  Call Extruder(8.25300)
  MoveL 4700 to (-39.1, 156.17, 78.65) mm, rotated rx -180 ry 0 rz 180 deg; joints [-141.891, 64.538, -73.427, 141.555, 83.016, 5.514]
  MoveL 4701 to (-39.1, 156.17, 78.65) mm, rotated rx -180 ry 0 rz 180 deg; joints [-141.891, 64.538, -73.427, 141.555, 83.016, 5.514]
  Call Extruder(8.43572)
  MoveL 4702 to (-39.22, 155.87, 78.65) mm, rotated rx -180 ry 0 rz 180 deg; joints [-141.96, 64.533, -73.433, 141.623, 83.001, 5.512]
  MoveL 4703 to (-39.22, 155.87, 78.65) mm, rotated rx -180 ry 0 rz 180 deg; joints [-141.96, 64.533, -73.433, 141.623, 83.001, 5.512]
  Call Extruder(8.61768)
  MoveL 4704 to (-39.35, 155.58, 78.65) mm, rotated rx -180 ry 0 rz 180 deg; joints [-142.029, 64.528, -73.439, 141.691, 82.986, 5.51]
  MoveL 4705 to (-39.35, 155.58, 78.65) mm, rotated rx -180 ry 0 rz 180 deg; joints [-142.029, 64.528, -73.439, 141.691, 82.986, 5.51]
  Call Extruder(8.76501)
  MoveL 4706 to (-39.44, 155.34, 78.65) mm, rotated rx -180 ry 0 rz 180 deg; joints [-142.085, 64.524, -73.444, 141.746, 82.973, 5.509]
  MoveL 4707 to (-39.44, 155.34, 78.65) mm, rotated rx -180 ry 0 rz 180 deg; joints [-142.085, 64.524, -73.444, 141.746, 82.973, 5.509]
  Call Extruder(8.87825)
  MoveL 4708 to (-39.5, 155.15, 78.65) mm, rotated rx -180 ry 0 rz 180 deg; joints [-142.127, 64.52, -73.449, 141.788, 82.963, 5.509]
  MoveL 4709 to (-39.5, 155.15, 78.65) mm, rotated rx -180 ry 0 rz 180 deg; joints [-142.127, 64.52, -73.449, 141.788, 82.963, 5.509]
  Call Extruder(8.99103)
  MoveL 4710 to (-39.56, 154.97, 78.65) mm, rotated rx -180 ry 0 rz 180 deg; joints [-142.169, 64.516, -73.453, 141.83, 82.952, 5.509]
  MoveL 4711 to (-39.56, 154.97, 78.65) mm, rotated rx -180 ry 0 rz 180 deg; joints [-142.169, 64.516, -73.453, 141.83, 82.952, 5.509]
  Call Extruder(9.10338)
  MoveL 4712 to (-39.62, 154.78, 78.65) mm, rotated rx 180 ry 0 rz 180 deg; joints [-142.212, 64.512, -73.458, 141.872, 82.941, 5.509]
  MoveL 4713 to (-39.62, 154.78, 78.65) mm, rotated rx 180 ry 0 rz 180 deg; joints [-142.212, 64.512, -73.458, 141.872, 82.941, 5.509]
  Call Extruder(9.21528)
  MoveL 4714 to (-39.68, 154.59, 78.65) mm, rotated rx 180 ry 0 rz -180 deg; joints [-142.254, 64.508, -73.462, 141.913, 82.931, 5.509]
  MoveL 4715 to (-39.68, 154.59, 78.65) mm, rotated rx 180 ry 0 rz -180 deg; joints [-142.254, 64.508, -73.462, 141.913, 82.931, 5.509]
  Call Extruder(9.33668)
  MoveL 4716 to (-39.75, 154.38, 78.65) mm, rotated rx 180 ry 0 rz 180 deg; joints [-142.3, 64.504, -73.467, 141.959, 82.919, 5.509]
  MoveL 4717 to (-39.75, 154.38, 78.65) mm, rotated rx 180 ry 0 rz 180 deg; joints [-142.3, 64.504, -73.467, 141.959, 82.919, 5.509]
  Call Extruder(9.46748)
  MoveL 4718 to (-39.81, 154.16, 78.65) mm, rotated rx -180 ry 0 rz 180 deg; joints [-142.35, 64.499, -73.473, 142.008, 82.906, 5.51]
  MoveL 4719 to (-39.81, 154.16, 78.65) mm, rotated rx -180 ry 0 rz 180 deg; joints [-142.35, 64.499, -73.473, 142.008, 82.906, 5.51]
  Call Extruder(9.59770)
  MoveL 4720 to (-39.88, 153.94, 78.65) mm, rotated rx 180 ry 0 rz 180 deg; joints [-142.399, 64.494, -73.478, 142.056, 82.893, 5.51]
  MoveL 4721 to (-39.88, 153.94, 78.65) mm, rotated rx 180 ry 0 rz 180 deg; joints [-142.399, 64.494, -73.478, 142.056, 82.893, 5.51]
  Call Extruder(9.72737)
  MoveL 4722 to (-39.95, 153.71, 78.65) mm, rotated rx -180 ry 0 rz 180 deg; joints [-142.449, 64.49, -73.484, 142.106, 82.88, 5.51]
  MoveL 4723 to (-39.95, 153.71, 78.65) mm, rotated rx -180 ry 0 rz 180 deg; joints [-142.449, 64.49, -73.484, 142.106, 82.88, 5.51]
  Call Extruder(9.85647)
  MoveL 4724 to (-40.02, 153.49, 78.65) mm, rotated rx 180 ry 0 rz -180 deg; joints [-142.498, 64.485, -73.49, 142.155, 82.867, 5.511]
  MoveL 4725 to (-40.02, 153.49, 78.65) mm, rotated rx 180 ry 0 rz -180 deg; joints [-142.498, 64.485, -73.49, 142.155, 82.867, 5.511]
  Call Extruder(9.97156)
  MoveL 4726 to (-40.06, 153.28, 78.65) mm, rotated rx 180 ry 0 rz 180 deg; joints [-142.541, 64.48, -73.496, 142.197, 82.854, 5.512]
  MoveL 4727 to (-40.06, 153.28, 78.65) mm, rotated rx 180 ry 0 rz 180 deg; joints [-142.541, 64.48, -73.496, 142.197, 82.854, 5.512]
  Call Extruder(10.08619)
  MoveL 4728 to (-40.11, 153.08, 78.65) mm, rotated rx -180 ry 0 rz 180 deg; joints [-142.584, 64.475, -73.501, 142.239, 82.841, 5.513]
  MoveL 4729 to (-40.11, 153.08, 78.65) mm, rotated rx -180 ry 0 rz 180 deg; joints [-142.584, 64.475, -73.501, 142.239, 82.841, 5.513]
  Call Extruder(10.20037)
  MoveL 4730 to (-40.15, 152.88, 78.65) mm, rotated rx -180 ry 0 rz 180 deg; joints [-142.627, 64.469, -73.507, 142.281, 82.829, 5.515]
  MoveL 4731 to (-40.15, 152.88, 78.65) mm, rotated rx -180 ry 0 rz 180 deg; joints [-142.627, 64.469, -73.507, 142.281, 82.829, 5.515]
  Call Extruder(10.31410)
  MoveL 4732 to (-40.2, 152.67, 78.65) mm, rotated rx -180 ry 0 rz 180 deg; joints [-142.671, 64.464, -73.513, 142.324, 82.816, 5.516]
  MoveL 4733 to (-40.2, 152.67, 78.65) mm, rotated rx -180 ry 0 rz 180 deg; joints [-142.671, 64.464, -73.513, 142.324, 82.816, 5.516]
  Call Extruder(10.43953)
  MoveL 4734 to (-40.24, 152.44, 78.65) mm, rotated rx 180 ry 0 rz 180 deg; joints [-142.718, 64.459, -73.52, 142.371, 82.801, 5.518]
  MoveL 4735 to (-40.24, 152.44, 78.65) mm, rotated rx 180 ry 0 rz 180 deg; joints [-142.718, 64.459, -73.52, 142.371, 82.801, 5.518]
  Call Extruder(10.57650)
  MoveL 4736 to (-40.29, 152.2, 78.65) mm, rotated rx -180 ry 0 rz -180 deg; joints [-142.77, 64.452, -73.527, 142.422, 82.785, 5.52]
  MoveL 4737 to (-40.29, 152.2, 78.65) mm, rotated rx -180 ry 0 rz -180 deg; joints [-142.77, 64.452, -73.527, 142.422, 82.785, 5.52]
  Call Extruder(10.71287)
  MoveL 4738 to (-40.34, 151.95, 78.65) mm, rotated rx 180 ry 0 rz 180 deg; joints [-142.822, 64.446, -73.535, 142.473, 82.769, 5.522]
  MoveL 4739 to (-40.34, 151.95, 78.65) mm, rotated rx 180 ry 0 rz 180 deg; joints [-142.822, 64.446, -73.535, 142.473, 82.769, 5.522]
  Call Extruder(10.84862)
  MoveL 4740 to (-40.39, 151.7, 78.65) mm, rotated rx 180 ry 0 rz 180 deg; joints [-142.874, 64.439, -73.542, 142.524, 82.753, 5.524]
  MoveL 4741 to (-40.39, 151.7, 78.65) mm, rotated rx 180 ry 0 rz 180 deg; joints [-142.874, 64.439, -73.542, 142.524, 82.753, 5.524]
  Call Extruder(10.98377)
  MoveL 4742 to (-40.44, 151.45, 78.65) mm, rotated rx -180 ry 0 rz 180 deg; joints [-142.926, 64.433, -73.55, 142.575, 82.737, 5.526]
  MoveL 4743 to (-40.44, 151.45, 78.65) mm, rotated rx -180 ry 0 rz 180 deg; joints [-142.926, 64.433, -73.55, 142.575, 82.737, 5.526]
  Call Extruder(11.11830)
  MoveL 4744 to (-40.49, 151.2, 78.65) mm, rotated rx -180 ry 0 rz 180 deg; joints [-142.978, 64.426, -73.557, 142.627, 82.721, 5.528]
  MoveL 4745 to (-40.49, 151.2, 78.65) mm, rotated rx -180 ry 0 rz 180 deg; joints [-142.978, 64.426, -73.557, 142.627, 82.721, 5.528]
  Call Extruder(11.25223)
  MoveL 4746 to (-40.54, 150.95, 78.65) mm, rotated rx -180 ry 0 rz 180 deg; joints [-143.031, 64.42, -73.565, 142.678, 82.705, 5.529]
  MoveL 4747 to (-40.54, 150.95, 78.65) mm, rotated rx -180 ry 0 rz 180 deg; joints [-143.031, 64.42, -73.565, 142.678, 82.705, 5.529]
  Call Extruder(11.40008)
  MoveL 4748 to (-40.59, 150.67, 78.65) mm, rotated rx -180 ry 0 rz -180 deg; joints [-143.088, 64.413, -73.573, 142.734, 82.687, 5.532]
  MoveL 4749 to (-40.59, 150.67, 78.65) mm, rotated rx -180 ry 0 rz -180 deg; joints [-143.088, 64.413, -73.573, 142.734, 82.687, 5.532]
  Call Extruder(11.56181)
  MoveL 4750 to (-40.64, 150.37, 78.65) mm, rotated rx 180 ry 0 rz -180 deg; joints [-143.15, 64.404, -73.583, 142.796, 82.667, 5.535]
  MoveL 4751 to (-40.64, 150.37, 78.65) mm, rotated rx 180 ry 0 rz -180 deg; joints [-143.15, 64.404, -73.583, 142.796, 82.667, 5.535]
  Call Extruder(11.72281)
  MoveL 4752 to (-40.69, 150.06, 78.65) mm, rotated rx 180 ry 0 rz -180 deg; joints [-143.213, 64.396, -73.592, 142.857, 82.646, 5.538]
  MoveL 4753 to (-40.69, 150.06, 78.65) mm, rotated rx 180 ry 0 rz -180 deg; joints [-143.213, 64.396, -73.592, 142.857, 82.646, 5.538]
  Call Extruder(11.88308)
  MoveL 4754 to (-40.74, 149.76, 78.65) mm, rotated rx -180 ry 0 rz 180 deg; joints [-143.276, 64.387, -73.602, 142.918, 82.626, 5.541]
  MoveL 4755 to (-40.74, 149.76, 78.65) mm, rotated rx -180 ry 0 rz 180 deg; joints [-143.276, 64.387, -73.602, 142.918, 82.626, 5.541]
  Call Extruder(12.04262)
  MoveL 4756 to (-40.78, 149.45, 78.65) mm, rotated rx -180 ry 0 rz 180 deg; joints [-143.338, 64.379, -73.611, 142.98, 82.605, 5.543]
  MoveL 4757 to (-40.78, 149.45, 78.65) mm, rotated rx -180 ry 0 rz 180 deg; joints [-143.338, 64.379, -73.611, 142.98, 82.605, 5.543]
  Call Extruder(12.20143)
  MoveL 4758 to (-40.83, 149.14, 78.65) mm, rotated rx -180 ry 0 rz 180 deg; joints [-143.401, 64.371, -73.621, 143.042, 82.585, 5.546]
  MoveL 4759 to (-40.83, 149.14, 78.65) mm, rotated rx -180 ry 0 rz 180 deg; joints [-143.401, 64.371, -73.621, 143.042, 82.585, 5.546]
  Call Extruder(12.38010)
  MoveL 4760 to (-40.88, 148.8, 78.65) mm, rotated rx 180 ry 0 rz -180 deg; joints [-143.471, 64.361, -73.632, 143.11, 82.561, 5.55]
  MoveL 4761 to (-40.88, 148.8, 78.65) mm, rotated rx 180 ry 0 rz -180 deg; joints [-143.471, 64.361, -73.632, 143.11, 82.561, 5.55]
  Call Extruder(12.57854)
  MoveL 4762 to (-40.92, 148.41, 78.65) mm, rotated rx -180 ry 0 rz 180 deg; joints [-143.549, 64.349, -73.645, 143.187, 82.535, 5.554]
  MoveL 4763 to (-40.92, 148.41, 78.65) mm, rotated rx -180 ry 0 rz 180 deg; joints [-143.549, 64.349, -73.645, 143.187, 82.535, 5.554]
  Call Extruder(12.77611)
  MoveL 4764 to (-40.97, 148.02, 78.65) mm, rotated rx -180 ry 0 rz -180 deg; joints [-143.627, 64.338, -73.658, 143.263, 82.508, 5.559]
  MoveL 4765 to (-40.97, 148.02, 78.65) mm, rotated rx -180 ry 0 rz -180 deg; joints [-143.627, 64.338, -73.658, 143.263, 82.508, 5.559]
  Call Extruder(12.97282)
  MoveL 4766 to (-41.02, 147.63, 78.65) mm, rotated rx -180 ry 0 rz -180 deg; joints [-143.705, 64.327, -73.671, 143.339, 82.481, 5.563]
  MoveL 4767 to (-41.02, 147.63, 78.65) mm, rotated rx -180 ry 0 rz -180 deg; joints [-143.705, 64.327, -73.671, 143.339, 82.481, 5.563]
  Call Extruder(13.16866)
  MoveL 4768 to (-41.06, 147.25, 78.65) mm, rotated rx -180 ry 0 rz 180 deg; joints [-143.783, 64.316, -73.683, 143.415, 82.454, 5.567]
  MoveL 4769 to (-41.06, 147.25, 78.65) mm, rotated rx -180 ry 0 rz 180 deg; joints [-143.783, 64.316, -73.683, 143.415, 82.454, 5.567]
  Call Extruder(13.46406)
  MoveL 4770 to (-41.11, 146.66, 78.65) mm, rotated rx -180 ry 0 rz -180 deg; joints [-143.899, 64.297, -73.704, 143.529, 82.412, 5.575]
  MoveL 4771 to (-41.11, 146.66, 78.65) mm, rotated rx -180 ry 0 rz -180 deg; joints [-143.899, 64.297, -73.704, 143.529, 82.412, 5.575]
  Call Extruder(13.75812)
  MoveL 4772 to (-41.16, 146.07, 78.65) mm, rotated rx -180 ry 0 rz 180 deg; joints [-144.015, 64.279, -73.724, 143.642, 82.369, 5.583]
  MoveL 4773 to (-41.16, 146.07, 78.65) mm, rotated rx -180 ry 0 rz 180 deg; joints [-144.015, 64.279, -73.724, 143.642, 82.369, 5.583]
  Call Extruder(14.05086)
  MoveL 4774 to (-41.2, 145.48, 78.65) mm, rotated rx -180 ry 0 rz 180 deg; joints [-144.131, 64.261, -73.744, 143.756, 82.327, 5.59]
  MoveL 4775 to (-41.2, 145.48, 78.65) mm, rotated rx -180 ry 0 rz 180 deg; joints [-144.131, 64.261, -73.744, 143.756, 82.327, 5.59]
  Call Extruder(14.62431)
  MoveL 4776 to (-41.25, 144.32, 78.65) mm, rotated rx -180 ry 0 rz -180 deg; joints [-144.355, 64.223, -73.786, 143.975, 82.241, 5.607]
  MoveL 4777 to (-41.25, 144.32, 78.65) mm, rotated rx -180 ry 0 rz -180 deg; joints [-144.355, 64.223, -73.786, 143.975, 82.241, 5.607]
  Call Extruder(15.33827)
  MoveL 4778 to (-41.29, 142.86, 78.65) mm, rotated rx -180 ry 0 rz 180 deg; joints [-144.635, 64.175, -73.839, 144.248, 82.131, 5.629]
  Call Extruder(57.40309)
  MoveL 4779 to (-41.29, 57.14, 78.65) mm, rotated rx -180 ry 0 rz 180 deg; joints [-164.153, 61.724, -76.018, 163.673, 76.26, 3.98]
  Call Extruder(57.83164)
  MoveL 4780 to (-41.27, 56.26, 78.65) mm, rotated rx -180 ry 0 rz 180 deg; joints [-164.382, 61.706, -76.031, 163.906, 76.215, 3.933]
  MoveL 4781 to (-41.27, 56.26, 78.65) mm, rotated rx -180 ry 0 rz 180 deg; joints [-164.382, 61.706, -76.031, 163.906, 76.215, 3.933]
  Call Extruder(58.40509)
  MoveL 4782 to (-41.22, 55.1, 78.65) mm, rotated rx 180 ry 0 rz 180 deg; joints [-164.686, 61.681, -76.049, 164.216, 76.153, 3.87]
  MoveL 4783 to (-41.22, 55.1, 78.65) mm, rotated rx 180 ry 0 rz 180 deg; joints [-164.686, 61.681, -76.049, 164.216, 76.153, 3.87]
  Call Extruder(58.83941)
  MoveL 4784 to (-41.18, 54.23, 78.65) mm, rotated rx 180 ry 0 rz -180 deg; joints [-164.915, 61.662, -76.063, 164.449, 76.105, 3.823]
  MoveL 4785 to (-41.18, 54.23, 78.65) mm, rotated rx 180 ry 0 rz -180 deg; joints [-164.915, 61.662, -76.063, 164.449, 76.105, 3.823]
  Call Extruder(59.13347)
  MoveL 4786 to (-41.13, 53.64, 78.65) mm, rotated rx 180 ry 0 rz 180 deg; joints [-165.068, 61.648, -76.073, 164.605, 76.072, 3.792]
  MoveL 4787 to (-41.13, 53.64, 78.65) mm, rotated rx 180 ry 0 rz 180 deg; joints [-165.068, 61.648, -76.073, 164.605, 76.072, 3.792]
  Call Extruder(59.42887)
  MoveL 4788 to (-41.09, 53.05, 78.65) mm, rotated rx 180 ry 0 rz 180 deg; joints [-165.222, 61.634, -76.083, 164.761, 76.039, 3.76]
  MoveL 4789 to (-41.09, 53.05, 78.65) mm, rotated rx 180 ry 0 rz 180 deg; joints [-165.222, 61.634, -76.083, 164.761, 76.039, 3.76]
  Call Extruder(59.67511)
  MoveL 4790 to (-41.04, 52.56, 78.65) mm, rotated rx 180 ry 0 rz -180 deg; joints [-165.349, 61.622, -76.091, 164.89, 76.011, 3.734]
  MoveL 4791 to (-41.04, 52.56, 78.65) mm, rotated rx 180 ry 0 rz -180 deg; joints [-165.349, 61.622, -76.091, 164.89, 76.011, 3.734]
  Call Extruder(59.87182)
  MoveL 4792 to (-40.99, 52.17, 78.65) mm, rotated rx -180 ry 0 rz 180 deg; joints [-165.449, 61.612, -76.099, 164.993, 75.987, 3.714]
  MoveL 4793 to (-40.99, 52.17, 78.65) mm, rotated rx -180 ry 0 rz 180 deg; joints [-165.449, 61.612, -76.099, 164.993, 75.987, 3.714]
  Call Extruder(60.06939)
  MoveL 4794 to (-40.95, 51.78, 78.65) mm, rotated rx -180 ry 0 rz 180 deg; joints [-165.549, 61.602, -76.106, 165.095, 75.964, 3.694]
  MoveL 4795 to (-40.95, 51.78, 78.65) mm, rotated rx -180 ry 0 rz 180 deg; joints [-165.549, 61.602, -76.106, 165.095, 75.964, 3.694]
  Call Extruder(60.26783)
  MoveL 4796 to (-40.9, 51.4, 78.65) mm, rotated rx 180 ry 0 rz 180 deg; joints [-165.65, 61.592, -76.113, 165.197, 75.941, 3.673]
  MoveL 4797 to (-40.9, 51.4, 78.65) mm, rotated rx 180 ry 0 rz 180 deg; joints [-165.65, 61.592, -76.113, 165.197, 75.941, 3.673]
  Call Extruder(60.46714)
  MoveL 4798 to (-40.86, 51.01, 78.65) mm, rotated rx -180 ry 0 rz -180 deg; joints [-165.751, 61.582, -76.12, 165.299, 75.918, 3.652]
  MoveL 4799 to (-40.86, 51.01, 78.65) mm, rotated rx -180 ry 0 rz -180 deg; joints [-165.751, 61.582, -76.12, 165.299, 75.918, 3.652]
  Call Extruder(60.62596)
  MoveL 4800 to (-40.81, 50.7, 78.65) mm, rotated rx 180 ry 0 rz -180 deg; joints [-165.829, 61.573, -76.126, 165.379, 75.899, 3.637]
  MoveL 4801 to (-40.81, 50.7, 78.65) mm, rotated rx 180 ry 0 rz -180 deg; joints [-165.829, 61.573, -76.126, 165.379, 75.899, 3.637]
  Call Extruder(60.78550)
  MoveL 4802 to (-40.76, 50.4, 78.65) mm, rotated rx 180 ry 0 rz 180 deg; joints [-165.908, 61.564, -76.132, 165.46, 75.88, 3.621]
  MoveL 4803 to (-40.76, 50.4, 78.65) mm, rotated rx 180 ry 0 rz 180 deg; joints [-165.908, 61.564, -76.132, 165.46, 75.88, 3.621]
  Call Extruder(60.94577)
  MoveL 4804 to (-40.71, 50.09, 78.65) mm, rotated rx 180 ry 0 rz 180 deg; joints [-165.987, 61.555, -76.138, 165.54, 75.861, 3.605]
  MoveL 4805 to (-40.71, 50.09, 78.65) mm, rotated rx 180 ry 0 rz 180 deg; joints [-165.987, 61.555, -76.138, 165.54, 75.861, 3.605]
  Call Extruder(61.10677)
  MoveL 4806 to (-40.66, 49.79, 78.65) mm, rotated rx -180 ry 0 rz -180 deg; joints [-166.066, 61.547, -76.144, 165.62, 75.841, 3.589]
  MoveL 4807 to (-40.66, 49.79, 78.65) mm, rotated rx -180 ry 0 rz -180 deg; joints [-166.066, 61.547, -76.144, 165.62, 75.841, 3.589]
  Call Extruder(61.26850)
  MoveL 4808 to (-40.61, 49.48, 78.65) mm, rotated rx 180 ry 0 rz 180 deg; joints [-166.145, 61.538, -76.15, 165.701, 75.822, 3.572]
  MoveL 4809 to (-40.61, 49.48, 78.65) mm, rotated rx 180 ry 0 rz 180 deg; joints [-166.145, 61.538, -76.15, 165.701, 75.822, 3.572]
  Call Extruder(61.43095)
  MoveL 4810 to (-40.57, 49.17, 78.65) mm, rotated rx 180 ry 0 rz -180 deg; joints [-166.224, 61.53, -76.156, 165.781, 75.803, 3.556]
  MoveL 4811 to (-40.57, 49.17, 78.65) mm, rotated rx 180 ry 0 rz -180 deg; joints [-166.224, 61.53, -76.156, 165.781, 75.803, 3.556]
  Call Extruder(61.56487)
  MoveL 4812 to (-40.52, 48.92, 78.65) mm, rotated rx 180 ry 0 rz 180 deg; joints [-166.288, 61.522, -76.161, 165.846, 75.787, 3.543]
  MoveL 4813 to (-40.52, 48.92, 78.65) mm, rotated rx 180 ry 0 rz 180 deg; joints [-166.288, 61.522, -76.161, 165.846, 75.787, 3.543]
  Call Extruder(61.69941)
  MoveL 4814 to (-40.47, 48.68, 78.65) mm, rotated rx -180 ry 0 rz -180 deg; joints [-166.352, 61.514, -76.167, 165.911, 75.77, 3.53]
  MoveL 4815 to (-40.47, 48.68, 78.65) mm, rotated rx -180 ry 0 rz -180 deg; joints [-166.352, 61.514, -76.167, 165.911, 75.77, 3.53]
  Call Extruder(61.83455)
  MoveL 4816 to (-40.42, 48.43, 78.65) mm, rotated rx 180 ry 0 rz -180 deg; joints [-166.416, 61.506, -76.172, 165.976, 75.754, 3.517]
  MoveL 4817 to (-40.42, 48.43, 78.65) mm, rotated rx 180 ry 0 rz -180 deg; joints [-166.416, 61.506, -76.172, 165.976, 75.754, 3.517]
  Call Extruder(61.97031)
  MoveL 4818 to (-40.37, 48.18, 78.65) mm, rotated rx -180 ry 0 rz 180 deg; joints [-166.48, 61.499, -76.177, 166.041, 75.737, 3.504]
  MoveL 4819 to (-40.37, 48.18, 78.65) mm, rotated rx -180 ry 0 rz 180 deg; joints [-166.48, 61.499, -76.177, 166.041, 75.737, 3.504]
  Call Extruder(62.10667)
  MoveL 4820 to (-40.32, 47.93, 78.65) mm, rotated rx -180 ry 0 rz 180 deg; joints [-166.544, 61.491, -76.183, 166.107, 75.721, 3.491]
  MoveL 4821 to (-40.32, 47.93, 78.65) mm, rotated rx -180 ry 0 rz 180 deg; joints [-166.544, 61.491, -76.183, 166.107, 75.721, 3.491]
  Call Extruder(62.24365)
  MoveL 4822 to (-40.27, 47.68, 78.65) mm, rotated rx -180 ry 0 rz 180 deg; joints [-166.608, 61.484, -76.188, 166.172, 75.704, 3.478]
  MoveL 4823 to (-40.27, 47.68, 78.65) mm, rotated rx -180 ry 0 rz 180 deg; joints [-166.608, 61.484, -76.188, 166.172, 75.704, 3.478]
  Call Extruder(62.38124)
  MoveL 4824 to (-40.22, 47.43, 78.65) mm, rotated rx -180 ry 0 rz 180 deg; joints [-166.673, 61.476, -76.193, 166.237, 75.688, 3.465]
  MoveL 4825 to (-40.22, 47.43, 78.65) mm, rotated rx -180 ry 0 rz 180 deg; joints [-166.673, 61.476, -76.193, 166.237, 75.688, 3.465]
  Call Extruder(62.49496)
  MoveL 4826 to (-40.17, 47.23, 78.65) mm, rotated rx -180 ry 0 rz 180 deg; joints [-166.725, 61.47, -76.197, 166.291, 75.674, 3.454]
  MoveL 4827 to (-40.17, 47.23, 78.65) mm, rotated rx -180 ry 0 rz 180 deg; joints [-166.725, 61.47, -76.197, 166.291, 75.674, 3.454]
  Call Extruder(62.60914)
  MoveL 4828 to (-40.13, 47.02, 78.65) mm, rotated rx 180 ry 0 rz 180 deg; joints [-166.778, 61.463, -76.202, 166.344, 75.66, 3.443]
  MoveL 4829 to (-40.13, 47.02, 78.65) mm, rotated rx 180 ry 0 rz 180 deg; joints [-166.778, 61.463, -76.202, 166.344, 75.66, 3.443]
  Call Extruder(62.72378)
  MoveL 4830 to (-40.08, 46.82, 78.65) mm, rotated rx 180 ry 0 rz -180 deg; joints [-166.83, 61.457, -76.206, 166.398, 75.646, 3.433]
  MoveL 4831 to (-40.08, 46.82, 78.65) mm, rotated rx 180 ry 0 rz -180 deg; joints [-166.83, 61.457, -76.206, 166.398, 75.646, 3.433]
  Call Extruder(62.83886)
  MoveL 4832 to (-40.04, 46.61, 78.65) mm, rotated rx -180 ry 0 rz 180 deg; joints [-166.883, 61.45, -76.211, 166.451, 75.633, 3.422]
  MoveL 4833 to (-40.04, 46.61, 78.65) mm, rotated rx -180 ry 0 rz 180 deg; joints [-166.883, 61.45, -76.211, 166.451, 75.633, 3.422]
  Call Extruder(62.96110)
  MoveL 4834 to (-39.98, 46.4, 78.65) mm, rotated rx -180 ry 0 rz -180 deg; joints [-166.937, 61.443, -76.216, 166.507, 75.617, 3.411]
  MoveL 4835 to (-39.98, 46.4, 78.65) mm, rotated rx -180 ry 0 rz -180 deg; joints [-166.937, 61.443, -76.216, 166.507, 75.617, 3.411]
  Call Extruder(63.09076)
  MoveL 4836 to (-39.92, 46.18, 78.65) mm, rotated rx -180 ry 0 rz 180 deg; joints [-166.994, 61.434, -76.222, 166.564, 75.6, 3.4]
  MoveL 4837 to (-39.92, 46.18, 78.65) mm, rotated rx -180 ry 0 rz 180 deg; joints [-166.994, 61.434, -76.222, 166.564, 75.6, 3.4]
  Call Extruder(63.22099)
  MoveL 4838 to (-39.85, 45.95, 78.65) mm, rotated rx -180 ry 0 rz 180 deg; joints [-167.051, 61.426, -76.227, 166.622, 75.583, 3.389]
  MoveL 4839 to (-39.85, 45.95, 78.65) mm, rotated rx -180 ry 0 rz 180 deg; joints [-167.051, 61.426, -76.227, 166.622, 75.583, 3.389]
  Call Extruder(63.35179)
  MoveL 4840 to (-39.78, 45.73, 78.65) mm, rotated rx 180 ry 0 rz -180 deg; joints [-167.107, 61.418, -76.233, 166.68, 75.566, 3.378]
  MoveL 4841 to (-39.78, 45.73, 78.65) mm, rotated rx 180 ry 0 rz -180 deg; joints [-167.107, 61.418, -76.233, 166.68, 75.566, 3.378]
  Call Extruder(63.48315)
  MoveL 4842 to (-39.71, 45.5, 78.65) mm, rotated rx 180 ry 0 rz 180 deg; joints [-167.164, 61.409, -76.239, 166.737, 75.549, 3.366]
  MoveL 4843 to (-39.71, 45.5, 78.65) mm, rotated rx 180 ry 0 rz 180 deg; joints [-167.164, 61.409, -76.239, 166.737, 75.549, 3.366]
  Call Extruder(63.59505)
  MoveL 4844 to (-39.65, 45.32, 78.65) mm, rotated rx -180 ry 0 rz -180 deg; joints [-167.212, 61.402, -76.244, 166.786, 75.534, 3.357]
  MoveL 4845 to (-39.65, 45.32, 78.65) mm, rotated rx -180 ry 0 rz -180 deg; joints [-167.212, 61.402, -76.244, 166.786, 75.534, 3.357]
  Call Extruder(63.70739)
  MoveL 4846 to (-39.59, 45.13, 78.65) mm, rotated rx -180 ry 0 rz -180 deg; joints [-167.26, 61.395, -76.249, 166.834, 75.52, 3.347]
  MoveL 4847 to (-39.59, 45.13, 78.65) mm, rotated rx -180 ry 0 rz -180 deg; joints [-167.26, 61.395, -76.249, 166.834, 75.52, 3.347]
  Call Extruder(63.82018)
  MoveL 4848 to (-39.53, 44.94, 78.65) mm, rotated rx -180 ry 0 rz -180 deg; joints [-167.307, 61.387, -76.254, 166.882, 75.505, 3.338]
  MoveL 4849 to (-39.53, 44.94, 78.65) mm, rotated rx -180 ry 0 rz -180 deg; joints [-167.307, 61.387, -76.254, 166.882, 75.505, 3.338]
  Call Extruder(63.93342)
  MoveL 4850 to (-39.47, 44.75, 78.65) mm, rotated rx 180 ry 0 rz 180 deg; joints [-167.355, 61.38, -76.259, 166.931, 75.49, 3.329]
  MoveL 4851 to (-39.47, 44.75, 78.65) mm, rotated rx 180 ry 0 rz 180 deg; joints [-167.355, 61.38, -76.259, 166.931, 75.49, 3.329]
  Call Extruder(64.04710)
  MoveL 4852 to (-39.41, 44.56, 78.65) mm, rotated rx -180 ry 0 rz 180 deg; joints [-167.403, 61.373, -76.264, 166.98, 75.475, 3.319]
  MoveL 4853 to (-39.41, 44.56, 78.65) mm, rotated rx -180 ry 0 rz 180 deg; joints [-167.403, 61.373, -76.264, 166.98, 75.475, 3.319]
  Call Extruder(64.22906)
  MoveL 4854 to (-39.29, 44.27, 78.65) mm, rotated rx -180 ry 0 rz -180 deg; joints [-167.475, 61.36, -76.272, 167.053, 75.45, 3.305]
  MoveL 4855 to (-39.29, 44.27, 78.65) mm, rotated rx -180 ry 0 rz -180 deg; joints [-167.475, 61.36, -76.272, 167.053, 75.45, 3.305]
  Call Extruder(64.41178)
  MoveL 4856 to (-39.17, 43.98, 78.65) mm, rotated rx -180 ry 0 rz 180 deg; joints [-167.548, 61.346, -76.281, 167.127, 75.424, 3.292]
  MoveL 4857 to (-39.17, 43.98, 78.65) mm, rotated rx -180 ry 0 rz 180 deg; joints [-167.548, 61.346, -76.281, 167.127, 75.424, 3.292]
  Call Extruder(64.58219)
  MoveL 4858 to (-39.05, 43.71, 78.65) mm, rotated rx -180 ry 0 rz -180 deg; joints [-167.615, 61.334, -76.29, 167.195, 75.4, 3.279]
  MoveL 4859 to (-39.05, 43.71, 78.65) mm, rotated rx -180 ry 0 rz -180 deg; joints [-167.615, 61.334, -76.29, 167.195, 75.4, 3.279]
  Call Extruder(64.74017)
  MoveL 4860 to (-38.94, 43.46, 78.65) mm, rotated rx -180 ry 0 rz -180 deg; joints [-167.677, 61.323, -76.297, 167.258, 75.378, 3.267]
  MoveL 4861 to (-38.94, 43.46, 78.65) mm, rotated rx -180 ry 0 rz -180 deg; joints [-167.677, 61.323, -76.297, 167.258, 75.378, 3.267]
  Call Extruder(64.89876)
  MoveL 4862 to (-38.84, 43.21, 78.65) mm, rotated rx 180 ry 0 rz 180 deg; joints [-167.739, 61.311, -76.305, 167.321, 75.356, 3.255]
  MoveL 4863 to (-38.84, 43.21, 78.65) mm, rotated rx 180 ry 0 rz 180 deg; joints [-167.739, 61.311, -76.305, 167.321, 75.356, 3.255]
  Call Extruder(65.10492)
  MoveL 4864 to (-38.66, 42.91, 78.65) mm, rotated rx -180 ry 0 rz -180 deg; joints [-167.813, 61.294, -76.316, 167.395, 75.324, 3.243]
  MoveL 4865 to (-38.66, 42.91, 78.65) mm, rotated rx -180 ry 0 rz -180 deg; joints [-167.813, 61.294, -76.316, 167.395, 75.324, 3.243]
  Call Extruder(65.31187)
  MoveL 4866 to (-38.49, 42.6, 78.65) mm, rotated rx 180 ry 0 rz 180 deg; joints [-167.886, 61.277, -76.328, 167.469, 75.292, 3.23]
  MoveL 4867 to (-38.49, 42.6, 78.65) mm, rotated rx 180 ry 0 rz 180 deg; joints [-167.886, 61.277, -76.328, 167.469, 75.292, 3.23]
  Call Extruder(65.51959)
  MoveL 4868 to (-38.31, 42.3, 78.65) mm, rotated rx 180 ry 0 rz 180 deg; joints [-167.96, 61.26, -76.339, 167.544, 75.26, 3.217]
  MoveL 4869 to (-38.31, 42.3, 78.65) mm, rotated rx 180 ry 0 rz 180 deg; joints [-167.96, 61.26, -76.339, 167.544, 75.26, 3.217]
  Call Extruder(65.72809)
  MoveL 4870 to (-38.14, 41.99, 78.65) mm, rotated rx -180 ry 0 rz -180 deg; joints [-168.033, 61.243, -76.351, 167.618, 75.228, 3.204]
  MoveL 4871 to (-38.14, 41.99, 78.65) mm, rotated rx -180 ry 0 rz -180 deg; joints [-168.033, 61.243, -76.351, 167.618, 75.228, 3.204]
  Call Extruder(65.90765)
  MoveL 4872 to (-37.96, 41.75, 78.65) mm, rotated rx -180 ry 0 rz -180 deg; joints [-168.091, 61.227, -76.361, 167.676, 75.199, 3.195]
  MoveL 4873 to (-37.96, 41.75, 78.65) mm, rotated rx -180 ry 0 rz -180 deg; joints [-168.091, 61.227, -76.361, 167.676, 75.199, 3.195]
  Call Extruder(66.24108)
  MoveL 4874 to (-37.63, 41.3, 78.65) mm, rotated rx -180 ry 0 rz 180 deg; joints [-168.197, 61.196, -76.381, 167.783, 75.144, 3.178]
  MoveL 4875 to (-37.63, 41.3, 78.65) mm, rotated rx -180 ry 0 rz 180 deg; joints [-168.197, 61.196, -76.381, 167.783, 75.144, 3.178]
  Call Extruder(66.57570)
  MoveL 4876 to (-37.3, 40.85, 78.65) mm, rotated rx 180 ry 0 rz -180 deg; joints [-168.304, 61.166, -76.401, 167.89, 75.089, 3.16]
  Call Extruder(67.40363)
  MoveL 4877 to (-36.39, 39.81, 78.65) mm, rotated rx -180 ry 0 rz 180 deg; joints [-168.541, 61.085, -76.454, 168.128, 74.946, 3.125]
  Call Extruder(68.23154)
  MoveL 4878 to (-35.35, 38.9, 78.65) mm, rotated rx -180 ry 0 rz -180 deg; joints [-168.739, 60.997, -76.51, 168.325, 74.793, 3.102]
  Call Extruder(68.39885)
  MoveL 4879 to (-35.13, 38.73, 78.65) mm, rotated rx 180 ry 0 rz 180 deg; joints [-168.773, 60.979, -76.522, 168.358, 74.761, 3.1]
  MoveL 4880 to (-35.13, 38.73, 78.65) mm, rotated rx 180 ry 0 rz 180 deg; joints [-168.773, 60.979, -76.522, 168.358, 74.761, 3.1]
  Call Extruder(68.73227)
  MoveL 4881 to (-34.68, 38.4, 78.65) mm, rotated rx 180 ry 0 rz 180 deg; joints [-168.84, 60.941, -76.546, 168.424, 74.698, 3.094]
  MoveL 4882 to (-34.68, 38.4, 78.65) mm, rotated rx 180 ry 0 rz 180 deg; joints [-168.84, 60.941, -76.546, 168.424, 74.698, 3.094]
  Call Extruder(69.06451)
  MoveL 4883 to (-34.23, 38.08, 78.65) mm, rotated rx -180 ry 0 rz -180 deg; joints [-168.908, 60.904, -76.569, 168.492, 74.634, 3.088]
  MoveL 4884 to (-34.23, 38.08, 78.65) mm, rotated rx -180 ry 0 rz -180 deg; joints [-168.908, 60.904, -76.569, 168.492, 74.634, 3.088]
  Call Extruder(69.18222)
  MoveL 4885 to (-34.05, 37.98, 78.65) mm, rotated rx -180 ry 0 rz -180 deg; joints [-168.927, 60.89, -76.578, 168.51, 74.611, 3.088]
  MoveL 4886 to (-34.05, 37.98, 78.65) mm, rotated rx -180 ry 0 rz -180 deg; joints [-168.927, 60.89, -76.578, 168.51, 74.611, 3.088]
  Call Extruder(69.38994)
  MoveL 4887 to (-33.75, 37.8, 78.65) mm, rotated rx 180 ry 0 rz 180 deg; joints [-168.96, 60.865, -76.593, 168.542, 74.57, 3.087]
  MoveL 4888 to (-33.75, 37.8, 78.65) mm, rotated rx 180 ry 0 rz 180 deg; joints [-168.96, 60.865, -76.593, 168.542, 74.57, 3.087]
  Call Extruder(69.59688)
  MoveL 4889 to (-33.45, 37.63, 78.65) mm, rotated rx -180 ry 0 rz 180 deg; joints [-168.993, 60.84, -76.609, 168.574, 74.529, 3.086]
  MoveL 4890 to (-33.45, 37.63, 78.65) mm, rotated rx -180 ry 0 rz 180 deg; joints [-168.993, 60.84, -76.609, 168.574, 74.529, 3.086]
  Call Extruder(69.80304)
  MoveL 4891 to (-33.14, 37.45, 78.65) mm, rotated rx -180 ry 0 rz -180 deg; joints [-169.026, 60.816, -76.624, 168.606, 74.488, 3.085]
  MoveL 4892 to (-33.14, 37.45, 78.65) mm, rotated rx -180 ry 0 rz -180 deg; joints [-169.026, 60.816, -76.624, 168.606, 74.488, 3.085]
  Call Extruder(69.98473)
  MoveL 4893 to (-32.87, 37.31, 78.65) mm, rotated rx 180 ry 0 rz 180 deg; joints [-169.052, 60.793, -76.638, 168.63, 74.451, 3.085]
  MoveL 4894 to (-32.87, 37.31, 78.65) mm, rotated rx 180 ry 0 rz 180 deg; joints [-169.052, 60.793, -76.638, 168.63, 74.451, 3.085]
  Call Extruder(70.14273)
  MoveL 4895 to (-32.62, 37.2, 78.65) mm, rotated rx 180 ry 0 rz 180 deg; joints [-169.068, 60.774, -76.65, 168.646, 74.419, 3.087]
  MoveL 4896 to (-32.62, 37.2, 78.65) mm, rotated rx 180 ry 0 rz 180 deg; joints [-169.068, 60.774, -76.65, 168.646, 74.419, 3.087]
  Call Extruder(70.30013)
  MoveL 4897 to (-32.37, 37.09, 78.65) mm, rotated rx -180 ry 0 rz 180 deg; joints [-169.085, 60.754, -76.662, 168.662, 74.387, 3.089]
  MoveL 4898 to (-32.37, 37.09, 78.65) mm, rotated rx -180 ry 0 rz 180 deg; joints [-169.085, 60.754, -76.662, 168.662, 74.387, 3.089]
  Call Extruder(70.48284)
  MoveL 4899 to (-32.07, 36.97, 78.65) mm, rotated rx -180 ry 0 rz 180 deg; joints [-169.104, 60.731, -76.676, 168.679, 74.349, 3.092]
  MoveL 4900 to (-32.07, 36.97, 78.65) mm, rotated rx -180 ry 0 rz 180 deg; joints [-169.104, 60.731, -76.676, 168.679, 74.349, 3.092]
  Call Extruder(70.66479)
  MoveL 4901 to (-31.78, 36.85, 78.65) mm, rotated rx -180 ry 0 rz -180 deg; joints [-169.122, 60.708, -76.69, 168.696, 74.312, 3.094]
  MoveL 4902 to (-31.78, 36.85, 78.65) mm, rotated rx -180 ry 0 rz -180 deg; joints [-169.122, 60.708, -76.69, 168.696, 74.312, 3.094]
  Call Extruder(70.81212)
  MoveL 4903 to (-31.54, 36.76, 78.65) mm, rotated rx -180 ry 0 rz -180 deg; joints [-169.135, 60.689, -76.702, 168.708, 74.281, 3.096]
  MoveL 4904 to (-31.54, 36.76, 78.65) mm, rotated rx -180 ry 0 rz -180 deg; joints [-169.135, 60.689, -76.702, 168.708, 74.281, 3.096]
  Call Extruder(70.92535)
  MoveL 4905 to (-31.35, 36.7, 78.65) mm, rotated rx -180 ry 0 rz 180 deg; joints [-169.143, 60.674, -76.711, 168.714, 74.258, 3.099]
  MoveL 4906 to (-31.35, 36.7, 78.65) mm, rotated rx -180 ry 0 rz 180 deg; joints [-169.143, 60.674, -76.711, 168.714, 74.258, 3.099]
  Call Extruder(71.03815)
  MoveL 4907 to (-31.17, 36.64, 78.65) mm, rotated rx -180 ry 0 rz 180 deg; joints [-169.15, 60.659, -76.72, 168.72, 74.234, 3.102]
  MoveL 4908 to (-31.17, 36.64, 78.65) mm, rotated rx -180 ry 0 rz 180 deg; joints [-169.15, 60.659, -76.72, 168.72, 74.234, 3.102]
  Call Extruder(71.15049)
  MoveL 4909 to (-30.98, 36.58, 78.65) mm, rotated rx -180 ry 0 rz 180 deg; joints [-169.157, 60.644, -76.729, 168.726, 74.21, 3.105]
  MoveL 4910 to (-30.98, 36.58, 78.65) mm, rotated rx -180 ry 0 rz 180 deg; joints [-169.157, 60.644, -76.729, 168.726, 74.21, 3.105]
  Call Extruder(71.26240)
  MoveL 4911 to (-30.79, 36.52, 78.65) mm, rotated rx -180 ry 0 rz 180 deg; joints [-169.164, 60.629, -76.737, 168.733, 74.187, 3.107]
  MoveL 4912 to (-30.79, 36.52, 78.65) mm, rotated rx -180 ry 0 rz 180 deg; joints [-169.164, 60.629, -76.737, 168.733, 74.187, 3.107]
  Call Extruder(71.38380)
  MoveL 4913 to (-30.58, 36.45, 78.65) mm, rotated rx 180 ry 0 rz 180 deg; joints [-169.172, 60.613, -76.747, 168.739, 74.161, 3.111]
  MoveL 4914 to (-30.58, 36.45, 78.65) mm, rotated rx 180 ry 0 rz 180 deg; joints [-169.172, 60.613, -76.747, 168.739, 74.161, 3.111]
  Call Extruder(71.51459)
  MoveL 4915 to (-30.36, 36.38, 78.65) mm, rotated rx -180 ry 0 rz -180 deg; joints [-169.179, 60.596, -76.758, 168.745, 74.133, 3.114]
  MoveL 4916 to (-30.36, 36.38, 78.65) mm, rotated rx -180 ry 0 rz -180 deg; joints [-169.179, 60.596, -76.758, 168.745, 74.133, 3.114]
  Call Extruder(71.64481)
  MoveL 4917 to (-30.14, 36.32, 78.65) mm, rotated rx -180 ry 0 rz -180 deg; joints [-169.186, 60.578, -76.768, 168.751, 74.106, 3.118]
  MoveL 4918 to (-30.14, 36.32, 78.65) mm, rotated rx -180 ry 0 rz -180 deg; joints [-169.186, 60.578, -76.768, 168.751, 74.106, 3.118]
  Call Extruder(71.77447)
  MoveL 4919 to (-29.91, 36.25, 78.65) mm, rotated rx -180 ry 0 rz -180 deg; joints [-169.193, 60.561, -76.778, 168.757, 74.078, 3.121]
  MoveL 4920 to (-29.91, 36.25, 78.65) mm, rotated rx -180 ry 0 rz -180 deg; joints [-169.193, 60.561, -76.778, 168.757, 74.078, 3.121]
  Call Extruder(71.90357)
  MoveL 4921 to (-29.69, 36.18, 78.65) mm, rotated rx -180 ry 0 rz -180 deg; joints [-169.201, 60.543, -76.789, 168.763, 74.05, 3.125]
  MoveL 4922 to (-29.69, 36.18, 78.65) mm, rotated rx -180 ry 0 rz -180 deg; joints [-169.201, 60.543, -76.789, 168.763, 74.05, 3.125]
  Call Extruder(72.01864)
  MoveL 4923 to (-29.48, 36.14, 78.65) mm, rotated rx -180 ry 0 rz 180 deg; joints [-169.202, 60.527, -76.798, 168.763, 74.025, 3.13]
  MoveL 4924 to (-29.48, 36.14, 78.65) mm, rotated rx -180 ry 0 rz 180 deg; joints [-169.202, 60.527, -76.798, 168.763, 74.025, 3.13]
  Call Extruder(72.13326)
  MoveL 4925 to (-29.28, 36.09, 78.65) mm, rotated rx -180 ry 0 rz 180 deg; joints [-169.204, 60.512, -76.807, 168.764, 74, 3.134]
  MoveL 4926 to (-29.28, 36.09, 78.65) mm, rotated rx -180 ry 0 rz 180 deg; joints [-169.204, 60.512, -76.807, 168.764, 74, 3.134]
  Call Extruder(72.24743)
  MoveL 4927 to (-29.08, 36.05, 78.65) mm, rotated rx -180 ry 0 rz 180 deg; joints [-169.206, 60.496, -76.817, 168.764, 73.976, 3.139]
  MoveL 4928 to (-29.08, 36.05, 78.65) mm, rotated rx -180 ry 0 rz 180 deg; joints [-169.206, 60.496, -76.817, 168.764, 73.976, 3.139]
  Call Extruder(72.36115)
  MoveL 4929 to (-28.87, 36, 78.65) mm, rotated rx 180 ry 0 rz 180 deg; joints [-169.207, 60.48, -76.826, 168.764, 73.951, 3.144]
  MoveL 4930 to (-28.87, 36, 78.65) mm, rotated rx 180 ry 0 rz 180 deg; joints [-169.207, 60.48, -76.826, 168.764, 73.951, 3.144]
  Call Extruder(72.48657)
  MoveL 4931 to (-28.65, 35.96, 78.65) mm, rotated rx -180 ry 0 rz 180 deg; joints [-169.208, 60.462, -76.836, 168.764, 73.924, 3.149]
  MoveL 4932 to (-28.65, 35.96, 78.65) mm, rotated rx -180 ry 0 rz 180 deg; joints [-169.208, 60.462, -76.836, 168.764, 73.924, 3.149]
  Call Extruder(72.62355)
  MoveL 4933 to (-28.4, 35.91, 78.65) mm, rotated rx -180 ry 0 rz 180 deg; joints [-169.209, 60.443, -76.847, 168.763, 73.894, 3.155]
  MoveL 4934 to (-28.4, 35.91, 78.65) mm, rotated rx -180 ry 0 rz 180 deg; joints [-169.209, 60.443, -76.847, 168.763, 73.894, 3.155]
  Call Extruder(72.75991)
  MoveL 4935 to (-28.15, 35.86, 78.65) mm, rotated rx 180 ry 0 rz 180 deg; joints [-169.21, 60.424, -76.859, 168.762, 73.864, 3.161]
  MoveL 4936 to (-28.15, 35.86, 78.65) mm, rotated rx 180 ry 0 rz 180 deg; joints [-169.21, 60.424, -76.859, 168.762, 73.864, 3.161]
  Call Extruder(72.89567)
  MoveL 4937 to (-27.9, 35.81, 78.65) mm, rotated rx -180 ry 0 rz -180 deg; joints [-169.21, 60.404, -76.87, 168.76, 73.834, 3.167]
  MoveL 4938 to (-27.9, 35.81, 78.65) mm, rotated rx -180 ry 0 rz -180 deg; joints [-169.21, 60.404, -76.87, 168.76, 73.834, 3.167]
  Call Extruder(73.03082)
  MoveL 4939 to (-27.65, 35.76, 78.65) mm, rotated rx -180 ry 0 rz 180 deg; joints [-169.211, 60.385, -76.881, 168.759, 73.804, 3.173]
  MoveL 4940 to (-27.65, 35.76, 78.65) mm, rotated rx -180 ry 0 rz 180 deg; joints [-169.211, 60.385, -76.881, 168.759, 73.804, 3.173]
  Call Extruder(73.16535)
  MoveL 4941 to (-27.4, 35.71, 78.65) mm, rotated rx -180 ry 0 rz -180 deg; joints [-169.212, 60.366, -76.892, 168.758, 73.774, 3.179]
  MoveL 4942 to (-27.4, 35.71, 78.65) mm, rotated rx -180 ry 0 rz -180 deg; joints [-169.212, 60.366, -76.892, 168.758, 73.774, 3.179]
  Call Extruder(73.29928)
  MoveL 4943 to (-27.15, 35.66, 78.65) mm, rotated rx 180 ry 0 rz -180 deg; joints [-169.212, 60.346, -76.903, 168.757, 73.744, 3.185]
  MoveL 4944 to (-27.15, 35.66, 78.65) mm, rotated rx 180 ry 0 rz -180 deg; joints [-169.212, 60.346, -76.903, 168.757, 73.744, 3.185]
  Call Extruder(73.44714)
  MoveL 4945 to (-26.87, 35.61, 78.65) mm, rotated rx -180 ry 0 rz 180 deg; joints [-169.211, 60.325, -76.916, 168.754, 73.711, 3.192]
  MoveL 4946 to (-26.87, 35.61, 78.65) mm, rotated rx -180 ry 0 rz 180 deg; joints [-169.211, 60.325, -76.916, 168.754, 73.711, 3.192]
  Call Extruder(73.60887)
  MoveL 4947 to (-26.57, 35.56, 78.65) mm, rotated rx -180 ry 0 rz 180 deg; joints [-169.208, 60.301, -76.929, 168.749, 73.675, 3.201]
  MoveL 4948 to (-26.57, 35.56, 78.65) mm, rotated rx -180 ry 0 rz 180 deg; joints [-169.208, 60.301, -76.929, 168.749, 73.675, 3.201]
  Call Extruder(73.76988)
  MoveL 4949 to (-26.26, 35.51, 78.65) mm, rotated rx -180 ry 0 rz -180 deg; joints [-169.205, 60.278, -76.943, 168.744, 73.638, 3.209]
  MoveL 4950 to (-26.26, 35.51, 78.65) mm, rotated rx -180 ry 0 rz -180 deg; joints [-169.205, 60.278, -76.943, 168.744, 73.638, 3.209]
  Call Extruder(73.93016)
  MoveL 4951 to (-25.96, 35.46, 78.65) mm, rotated rx 180 ry 0 rz 180 deg; joints [-169.202, 60.254, -76.956, 168.739, 73.602, 3.217]
  MoveL 4952 to (-25.96, 35.46, 78.65) mm, rotated rx 180 ry 0 rz 180 deg; joints [-169.202, 60.254, -76.956, 168.739, 73.602, 3.217]
  Call Extruder(74.08971)
  MoveL 4953 to (-25.65, 35.42, 78.65) mm, rotated rx -180 ry 0 rz -180 deg; joints [-169.199, 60.23, -76.969, 168.733, 73.566, 3.226]
  MoveL 4954 to (-25.65, 35.42, 78.65) mm, rotated rx -180 ry 0 rz -180 deg; joints [-169.199, 60.23, -76.969, 168.733, 73.566, 3.226]
  Call Extruder(74.24853)
  MoveL 4955 to (-25.34, 35.37, 78.65) mm, rotated rx -180 ry 0 rz -180 deg; joints [-169.196, 60.206, -76.983, 168.728, 73.53, 3.234]
  MoveL 4956 to (-25.34, 35.37, 78.65) mm, rotated rx -180 ry 0 rz -180 deg; joints [-169.196, 60.206, -76.983, 168.728, 73.53, 3.234]
  Call Extruder(74.42720)
  MoveL 4957 to (-25, 35.32, 78.65) mm, rotated rx -180 ry 0 rz 180 deg; joints [-169.191, 60.18, -76.998, 168.72, 73.489, 3.244]
  MoveL 4958 to (-25, 35.32, 78.65) mm, rotated rx -180 ry 0 rz 180 deg; joints [-169.191, 60.18, -76.998, 168.72, 73.489, 3.244]
  Call Extruder(74.62564)
  MoveL 4959 to (-24.61, 35.28, 78.65) mm, rotated rx -180 ry 0 rz -180 deg; joints [-169.182, 60.15, -77.014, 168.708, 73.444, 3.256]
  MoveL 4960 to (-24.61, 35.28, 78.65) mm, rotated rx -180 ry 0 rz -180 deg; joints [-169.182, 60.15, -77.014, 168.708, 73.444, 3.256]
  Call Extruder(74.82322)
  MoveL 4961 to (-24.22, 35.23, 78.65) mm, rotated rx -180 ry 0 rz 180 deg; joints [-169.174, 60.12, -77.031, 168.697, 73.399, 3.268]
  MoveL 4962 to (-24.22, 35.23, 78.65) mm, rotated rx -180 ry 0 rz 180 deg; joints [-169.174, 60.12, -77.031, 168.697, 73.399, 3.268]
  Call Extruder(75.01993)
  MoveL 4963 to (-23.84, 35.18, 78.65) mm, rotated rx -180 ry 0 rz -180 deg; joints [-169.166, 60.09, -77.047, 168.685, 73.353, 3.28]
  MoveL 4964 to (-23.84, 35.18, 78.65) mm, rotated rx -180 ry 0 rz -180 deg; joints [-169.166, 60.09, -77.047, 168.685, 73.353, 3.28]
  Call Extruder(75.21577)
  MoveL 4965 to (-23.45, 35.14, 78.65) mm, rotated rx -180 ry 0 rz -180 deg; joints [-169.157, 60.059, -77.064, 168.674, 73.308, 3.293]
  MoveL 4966 to (-23.45, 35.14, 78.65) mm, rotated rx -180 ry 0 rz -180 deg; joints [-169.157, 60.059, -77.064, 168.674, 73.308, 3.293]
  Call Extruder(75.51116)
  MoveL 4967 to (-22.86, 35.09, 78.65) mm, rotated rx -180 ry 0 rz -180 deg; joints [-169.137, 60.014, -77.089, 168.649, 73.24, 3.313]
  MoveL 4968 to (-22.86, 35.09, 78.65) mm, rotated rx -180 ry 0 rz -180 deg; joints [-169.137, 60.014, -77.089, 168.649, 73.24, 3.313]
  Call Extruder(75.80522)
  MoveL 4969 to (-22.27, 35.04, 78.65) mm, rotated rx 180 ry 0 rz 180 deg; joints [-169.117, 59.968, -77.113, 168.623, 73.173, 3.334]
  MoveL 4970 to (-22.27, 35.04, 78.65) mm, rotated rx 180 ry 0 rz 180 deg; joints [-169.117, 59.968, -77.113, 168.623, 73.173, 3.334]
  Call Extruder(76.09795)
  MoveL 4971 to (-21.68, 35, 78.65) mm, rotated rx 180 ry 0 rz 180 deg; joints [-169.096, 59.923, -77.138, 168.598, 73.105, 3.354]
  MoveL 4972 to (-21.68, 35, 78.65) mm, rotated rx 180 ry 0 rz 180 deg; joints [-169.096, 59.923, -77.138, 168.598, 73.105, 3.354]
  Call Extruder(76.67140)
  MoveL 4973 to (-20.52, 34.95, 78.65) mm, rotated rx -180 ry 0 rz -180 deg; joints [-169.042, 59.833, -77.185, 168.533, 72.974, 3.399]
  MoveL 4974 to (-20.52, 34.95, 78.65) mm, rotated rx -180 ry 0 rz -180 deg; joints [-169.042, 59.833, -77.185, 168.533, 72.974, 3.399]
  Call Extruder(77.38537)
  MoveL 4975 to (-19.06, 34.91, 78.65) mm, rotated rx -180 ry 0 rz -180 deg; joints [-168.967, 59.72, -77.244, 168.445, 72.81, 3.458]
  Call Extruder(194.23211)
  MoveL 4976 to (219.06, 34.91, 78.65) mm, rotated rx 180 ry 0 rz 180 deg; joints [-30.588, 49.086, -79.42, 34.406, 115.77, 16.581]
  Call Extruder(194.66067)
  MoveL 4977 to (219.94, 34.93, 78.65) mm, rotated rx -180 ry 0 rz 180 deg; joints [-30.233, 49.168, -79.422, 34.007, 115.805, 16.367]
  MoveL 4978 to (219.94, 34.93, 78.65) mm, rotated rx -180 ry 0 rz 180 deg; joints [-30.233, 49.168, -79.422, 34.007, 115.805, 16.367]
  Call Extruder(195.23412)
  MoveL 4979 to (221.1, 34.97, 78.65) mm, rotated rx -180 ry 0 rz 180 deg; joints [-29.789, 49.277, -79.424, 33.504, 115.84, 16.094]
  MoveL 4980 to (221.1, 34.97, 78.65) mm, rotated rx -180 ry 0 rz 180 deg; joints [-29.789, 49.277, -79.424, 33.504, 115.84, 16.094]
  Call Extruder(195.66843)
  MoveL 4981 to (221.97, 35.02, 78.65) mm, rotated rx -180 ry 0 rz 180 deg; joints [-29.47, 49.361, -79.425, 33.142, 115.859, 15.896]
  MoveL 4982 to (221.97, 35.02, 78.65) mm, rotated rx -180 ry 0 rz 180 deg; joints [-29.47, 49.361, -79.425, 33.142, 115.859, 15.896]
  Call Extruder(195.96249)
  MoveL 4983 to (222.56, 35.07, 78.65) mm, rotated rx -180 ry 0 rz 180 deg; joints [-29.272, 49.418, -79.426, 32.915, 115.866, 15.769]
  MoveL 4984 to (222.56, 35.07, 78.65) mm, rotated rx -180 ry 0 rz 180 deg; joints [-29.272, 49.418, -79.426, 32.915, 115.866, 15.769]
  Call Extruder(196.25788)
  MoveL 4985 to (223.15, 35.11, 78.65) mm, rotated rx -180 ry 0 rz 180 deg; joints [-29.075, 49.475, -79.427, 32.689, 115.872, 15.643]
  MoveL 4986 to (223.15, 35.11, 78.65) mm, rotated rx -180 ry 0 rz 180 deg; joints [-29.075, 49.475, -79.427, 32.689, 115.872, 15.643]
  Call Extruder(196.50411)
  MoveL 4987 to (223.64, 35.16, 78.65) mm, rotated rx -180 ry 0 rz 180 deg; joints [-28.92, 49.522, -79.427, 32.511, 115.874, 15.543]
  MoveL 4988 to (223.64, 35.16, 78.65) mm, rotated rx -180 ry 0 rz 180 deg; joints [-28.92, 49.522, -79.427, 32.511, 115.874, 15.543]
  Call Extruder(196.70082)
  MoveL 4989 to (224.03, 35.21, 78.65) mm, rotated rx -180 ry 0 rz 180 deg; joints [-28.804, 49.561, -79.427, 32.377, 115.872, 15.466]
  MoveL 4990 to (224.03, 35.21, 78.65) mm, rotated rx -180 ry 0 rz 180 deg; joints [-28.804, 49.561, -79.427, 32.377, 115.872, 15.466]
  Call Extruder(196.89839)
  MoveL 4991 to (224.42, 35.25, 78.65) mm, rotated rx -180 ry 0 rz 180 deg; joints [-28.69, 49.599, -79.428, 32.245, 115.871, 15.39]
  MoveL 4992 to (224.42, 35.25, 78.65) mm, rotated rx -180 ry 0 rz 180 deg; joints [-28.69, 49.599, -79.428, 32.245, 115.871, 15.39]
  Call Extruder(197.09684)
  MoveL 4993 to (224.8, 35.3, 78.65) mm, rotated rx -180 ry 0 rz 180 deg; joints [-28.577, 49.637, -79.428, 32.114, 115.868, 15.314]
  MoveL 4994 to (224.8, 35.3, 78.65) mm, rotated rx -180 ry 0 rz 180 deg; joints [-28.577, 49.637, -79.428, 32.114, 115.868, 15.314]
  Call Extruder(197.29615)
  MoveL 4995 to (225.19, 35.34, 78.65) mm, rotated rx 180 ry 0 rz -180 deg; joints [-28.465, 49.676, -79.428, 31.984, 115.865, 15.24]
  MoveL 4996 to (225.19, 35.34, 78.65) mm, rotated rx 180 ry 0 rz -180 deg; joints [-28.465, 49.676, -79.428, 31.984, 115.865, 15.24]
  Call Extruder(197.45497)
  MoveL 4997 to (225.5, 35.39, 78.65) mm, rotated rx -180 ry 0 rz -180 deg; joints [-28.385, 49.707, -79.428, 31.891, 115.86, 15.184]
  MoveL 4998 to (225.5, 35.39, 78.65) mm, rotated rx -180 ry 0 rz -180 deg; joints [-28.385, 49.707, -79.428, 31.891, 115.86, 15.184]
  Call Extruder(197.61451)
  MoveL 4999 to (225.8, 35.44, 78.65) mm, rotated rx -180 ry 0 rz 180 deg; joints [-28.307, 49.737, -79.428, 31.798, 115.855, 15.129]
  MoveL 5000 to (225.8, 35.44, 78.65) mm, rotated rx -180 ry 0 rz 180 deg; joints [-28.307, 49.737, -79.428, 31.798, 115.855, 15.129]
  Call Extruder(197.77479)
  MoveL 5001 to (226.11, 35.49, 78.65) mm, rotated rx -180 ry 0 rz -180 deg; joints [-28.228, 49.768, -79.428, 31.707, 115.849, 15.075]
  MoveL 5002 to (226.11, 35.49, 78.65) mm, rotated rx -180 ry 0 rz -180 deg; joints [-28.228, 49.768, -79.428, 31.707, 115.849, 15.075]
  Call Extruder(197.93579)
  MoveL 5003 to (226.41, 35.54, 78.65) mm, rotated rx -180 ry 0 rz 180 deg; joints [-28.151, 49.799, -79.428, 31.616, 115.843, 15.021]
  MoveL 5004 to (226.41, 35.54, 78.65) mm, rotated rx -180 ry 0 rz 180 deg; joints [-28.151, 49.799, -79.428, 31.616, 115.843, 15.021]
  Call Extruder(198.09752)
  MoveL 5005 to (226.72, 35.59, 78.65) mm, rotated rx 180 ry 0 rz 180 deg; joints [-28.074, 49.83, -79.428, 31.525, 115.836, 14.967]
  MoveL 5006 to (226.72, 35.59, 78.65) mm, rotated rx 180 ry 0 rz 180 deg; joints [-28.074, 49.83, -79.428, 31.525, 115.836, 14.967]
  Call Extruder(198.25998)
  MoveL 5007 to (227.03, 35.64, 78.65) mm, rotated rx -180 ry 0 rz -180 deg; joints [-27.998, 49.861, -79.428, 31.436, 115.83, 14.913]
  MoveL 5008 to (227.03, 35.64, 78.65) mm, rotated rx -180 ry 0 rz -180 deg; joints [-27.998, 49.861, -79.428, 31.436, 115.83, 14.913]
  Call Extruder(198.39391)
  MoveL 5009 to (227.27, 35.68, 78.65) mm, rotated rx -180 ry 0 rz 180 deg; joints [-27.942, 49.886, -79.428, 31.37, 115.822, 14.872]
  MoveL 5010 to (227.27, 35.68, 78.65) mm, rotated rx -180 ry 0 rz 180 deg; joints [-27.942, 49.886, -79.428, 31.37, 115.822, 14.872]
  Call Extruder(198.52845)
  MoveL 5011 to (227.52, 35.73, 78.65) mm, rotated rx -180 ry 0 rz 180 deg; joints [-27.888, 49.912, -79.428, 31.305, 115.814, 14.832]
  MoveL 5012 to (227.52, 35.73, 78.65) mm, rotated rx -180 ry 0 rz 180 deg; joints [-27.888, 49.912, -79.428, 31.305, 115.814, 14.832]
  Call Extruder(198.66359)
  MoveL 5013 to (227.77, 35.78, 78.65) mm, rotated rx 180 ry 0 rz 180 deg; joints [-27.834, 49.938, -79.428, 31.24, 115.806, 14.792]
  MoveL 5014 to (227.77, 35.78, 78.65) mm, rotated rx 180 ry 0 rz 180 deg; joints [-27.834, 49.938, -79.428, 31.24, 115.806, 14.792]
  Call Extruder(198.79935)
  MoveL 5015 to (228.02, 35.83, 78.65) mm, rotated rx -180 ry 0 rz 180 deg; joints [-27.78, 49.963, -79.427, 31.176, 115.797, 14.752]
  MoveL 5016 to (228.02, 35.83, 78.65) mm, rotated rx -180 ry 0 rz 180 deg; joints [-27.78, 49.963, -79.427, 31.176, 115.797, 14.752]
  Call Extruder(198.93572)
  MoveL 5017 to (228.27, 35.88, 78.65) mm, rotated rx -180 ry 0 rz 180 deg; joints [-27.726, 49.989, -79.427, 31.112, 115.789, 14.712]
  MoveL 5018 to (228.27, 35.88, 78.65) mm, rotated rx -180 ry 0 rz 180 deg; joints [-27.726, 49.989, -79.427, 31.112, 115.789, 14.712]
  Call Extruder(199.07270)
  MoveL 5019 to (228.52, 35.93, 78.65) mm, rotated rx -180 ry 0 rz 180 deg; joints [-27.673, 50.014, -79.427, 31.048, 115.781, 14.672]
  MoveL 5020 to (228.52, 35.93, 78.65) mm, rotated rx -180 ry 0 rz 180 deg; joints [-27.673, 50.014, -79.427, 31.048, 115.781, 14.672]
  Call Extruder(199.21029)
  MoveL 5021 to (228.77, 35.98, 78.65) mm, rotated rx 180 ry 0 rz 180 deg; joints [-27.62, 50.04, -79.427, 30.985, 115.772, 14.633]
  MoveL 5022 to (228.77, 35.98, 78.65) mm, rotated rx 180 ry 0 rz 180 deg; joints [-27.62, 50.04, -79.427, 30.985, 115.772, 14.633]
  Call Extruder(199.32400)
  MoveL 5023 to (228.97, 36.03, 78.65) mm, rotated rx -180 ry 0 rz 180 deg; joints [-27.579, 50.061, -79.427, 30.936, 115.764, 14.601]
  MoveL 5024 to (228.97, 36.03, 78.65) mm, rotated rx -180 ry 0 rz 180 deg; joints [-27.579, 50.061, -79.427, 30.936, 115.764, 14.601]
  Call Extruder(199.43818)
  MoveL 5025 to (229.18, 36.07, 78.65) mm, rotated rx -180 ry 0 rz 180 deg; joints [-27.539, 50.082, -79.426, 30.887, 115.756, 14.57]
  MoveL 5026 to (229.18, 36.07, 78.65) mm, rotated rx -180 ry 0 rz 180 deg; joints [-27.539, 50.082, -79.426, 30.887, 115.756, 14.57]
  Call Extruder(199.55280)
  MoveL 5027 to (229.38, 36.12, 78.65) mm, rotated rx -180 ry 0 rz -180 deg; joints [-27.499, 50.103, -79.426, 30.839, 115.747, 14.539]
  MoveL 5028 to (229.38, 36.12, 78.65) mm, rotated rx -180 ry 0 rz -180 deg; joints [-27.499, 50.103, -79.426, 30.839, 115.747, 14.539]
  Call Extruder(199.66788)
  MoveL 5029 to (229.59, 36.16, 78.65) mm, rotated rx 180 ry 0 rz 180 deg; joints [-27.458, 50.124, -79.426, 30.79, 115.739, 14.509]
  MoveL 5030 to (229.59, 36.16, 78.65) mm, rotated rx 180 ry 0 rz 180 deg; joints [-27.458, 50.124, -79.426, 30.79, 115.739, 14.509]
  Call Extruder(199.79011)
  MoveL 5031 to (229.8, 36.22, 78.65) mm, rotated rx 180 ry 0 rz 180 deg; joints [-27.423, 50.147, -79.426, 30.746, 115.728, 14.479]
  MoveL 5032 to (229.8, 36.22, 78.65) mm, rotated rx 180 ry 0 rz 180 deg; joints [-27.423, 50.147, -79.426, 30.746, 115.728, 14.479]
  Call Extruder(199.91978)
  MoveL 5033 to (230.02, 36.28, 78.65) mm, rotated rx 180 ry 0 rz -180 deg; joints [-27.392, 50.171, -79.425, 30.707, 115.715, 14.451]
  MoveL 5034 to (230.02, 36.28, 78.65) mm, rotated rx 180 ry 0 rz -180 deg; joints [-27.392, 50.171, -79.425, 30.707, 115.715, 14.451]
  Call Extruder(200.05001)
  MoveL 5035 to (230.25, 36.35, 78.65) mm, rotated rx -180 ry 0 rz 180 deg; joints [-27.361, 50.195, -79.425, 30.668, 115.702, 14.422]
  MoveL 5036 to (230.25, 36.35, 78.65) mm, rotated rx -180 ry 0 rz 180 deg; joints [-27.361, 50.195, -79.425, 30.668, 115.702, 14.422]
  Call Extruder(200.18080)
  MoveL 5037 to (230.47, 36.42, 78.65) mm, rotated rx 180 ry 0 rz 180 deg; joints [-27.33, 50.219, -79.425, 30.628, 115.689, 14.394]
  MoveL 5038 to (230.47, 36.42, 78.65) mm, rotated rx 180 ry 0 rz 180 deg; joints [-27.33, 50.219, -79.425, 30.628, 115.689, 14.394]
  Call Extruder(200.31217)
  MoveL 5039 to (230.69, 36.49, 78.65) mm, rotated rx -180 ry 0 rz 180 deg; joints [-27.299, 50.243, -79.424, 30.589, 115.675, 14.366]
  MoveL 5040 to (230.69, 36.49, 78.65) mm, rotated rx -180 ry 0 rz 180 deg; joints [-27.299, 50.243, -79.424, 30.589, 115.675, 14.366]
  Call Extruder(200.42119)
  MoveL 5041 to (230.88, 36.55, 78.65) mm, rotated rx -180 ry 0 rz 180 deg; joints [-27.277, 50.263, -79.424, 30.561, 115.663, 14.344]
  MoveL 5042 to (230.88, 36.55, 78.65) mm, rotated rx -180 ry 0 rz 180 deg; joints [-27.277, 50.263, -79.424, 30.561, 115.663, 14.344]
  Call Extruder(200.53270)
  MoveL 5043 to (231.06, 36.61, 78.65) mm, rotated rx -180 ry 0 rz 180 deg; joints [-27.254, 50.283, -79.424, 30.531, 115.651, 14.322]
  MoveL 5044 to (231.06, 36.61, 78.65) mm, rotated rx -180 ry 0 rz 180 deg; joints [-27.254, 50.283, -79.424, 30.531, 115.651, 14.322]
  Call Extruder(200.64671)
  MoveL 5045 to (231.26, 36.67, 78.65) mm, rotated rx -180 ry 0 rz -180 deg; joints [-27.231, 50.304, -79.423, 30.501, 115.639, 14.299]
  MoveL 5046 to (231.26, 36.67, 78.65) mm, rotated rx -180 ry 0 rz -180 deg; joints [-27.231, 50.304, -79.423, 30.501, 115.639, 14.299]
  Call Extruder(200.76118)
  MoveL 5047 to (231.45, 36.73, 78.65) mm, rotated rx 180 ry 0 rz 180 deg; joints [-27.208, 50.325, -79.423, 30.471, 115.626, 14.277]
  MoveL 5048 to (231.45, 36.73, 78.65) mm, rotated rx 180 ry 0 rz 180 deg; joints [-27.208, 50.325, -79.423, 30.471, 115.626, 14.277]
  Call Extruder(200.87611)
  MoveL 5049 to (231.64, 36.79, 78.65) mm, rotated rx -180 ry 0 rz 180 deg; joints [-27.185, 50.345, -79.422, 30.441, 115.614, 14.254]
  MoveL 5050 to (231.64, 36.79, 78.65) mm, rotated rx -180 ry 0 rz 180 deg; joints [-27.185, 50.345, -79.422, 30.441, 115.614, 14.254]
  Call Extruder(201.05806)
  MoveL 5051 to (231.93, 36.91, 78.65) mm, rotated rx 180 ry 0 rz 180 deg; joints [-27.167, 50.378, -79.422, 30.414, 115.589, 14.227]
  MoveL 5052 to (231.93, 36.91, 78.65) mm, rotated rx 180 ry 0 rz 180 deg; joints [-27.167, 50.378, -79.422, 30.414, 115.589, 14.227]
  Call Extruder(201.24078)
  MoveL 5053 to (232.22, 37.04, 78.65) mm, rotated rx 180 ry 0 rz -180 deg; joints [-27.149, 50.411, -79.421, 30.386, 115.565, 14.2]
  MoveL 5054 to (232.22, 37.04, 78.65) mm, rotated rx 180 ry 0 rz -180 deg; joints [-27.149, 50.411, -79.421, 30.386, 115.565, 14.2]
  Call Extruder(201.41120)
  MoveL 5055 to (232.49, 37.15, 78.65) mm, rotated rx 180 ry 0 rz 180 deg; joints [-27.133, 50.441, -79.42, 30.362, 115.542, 14.175]
  MoveL 5056 to (232.49, 37.15, 78.65) mm, rotated rx 180 ry 0 rz 180 deg; joints [-27.133, 50.441, -79.42, 30.362, 115.542, 14.175]
  Call Extruder(201.56919)
  MoveL 5057 to (232.74, 37.26, 78.65) mm, rotated rx 180 ry 0 rz -180 deg; joints [-27.121, 50.469, -79.42, 30.341, 115.52, 14.153]
  MoveL 5058 to (232.74, 37.26, 78.65) mm, rotated rx 180 ry 0 rz -180 deg; joints [-27.121, 50.469, -79.42, 30.341, 115.52, 14.153]
  Call Extruder(201.72780)
  MoveL 5059 to (232.99, 37.36, 78.65) mm, rotated rx -180 ry 0 rz 180 deg; joints [-27.108, 50.498, -79.419, 30.32, 115.498, 14.131]
  MoveL 5060 to (232.99, 37.36, 78.65) mm, rotated rx -180 ry 0 rz 180 deg; joints [-27.108, 50.498, -79.419, 30.32, 115.498, 14.131]
  Call Extruder(201.93396)
  MoveL 5061 to (233.29, 37.54, 78.65) mm, rotated rx -180 ry 0 rz 180 deg; joints [-27.12, 50.534, -79.418, 30.324, 115.463, 14.116]
  MoveL 5062 to (233.29, 37.54, 78.65) mm, rotated rx -180 ry 0 rz 180 deg; joints [-27.12, 50.534, -79.418, 30.324, 115.463, 14.116]
  Call Extruder(202.14091)
  MoveL 5063 to (233.6, 37.71, 78.65) mm, rotated rx -180 ry 0 rz 180 deg; joints [-27.132, 50.571, -79.417, 30.329, 115.428, 14.101]
  MoveL 5064 to (233.6, 37.71, 78.65) mm, rotated rx -180 ry 0 rz 180 deg; joints [-27.132, 50.571, -79.417, 30.329, 115.428, 14.101]
  Call Extruder(202.34863)
  MoveL 5065 to (233.9, 37.89, 78.65) mm, rotated rx 180 ry 0 rz 180 deg; joints [-27.144, 50.607, -79.416, 30.332, 115.393, 14.085]
  MoveL 5066 to (233.9, 37.89, 78.65) mm, rotated rx 180 ry 0 rz 180 deg; joints [-27.144, 50.607, -79.416, 30.332, 115.393, 14.085]
  Call Extruder(202.55713)
  MoveL 5067 to (234.21, 38.07, 78.65) mm, rotated rx -180 ry 0 rz 180 deg; joints [-27.156, 50.643, -79.415, 30.337, 115.357, 14.07]
  MoveL 5068 to (234.21, 38.07, 78.65) mm, rotated rx -180 ry 0 rz 180 deg; joints [-27.156, 50.643, -79.415, 30.337, 115.357, 14.07]
  Call Extruder(202.73668)
  MoveL 5069 to (234.45, 38.24, 78.65) mm, rotated rx -180 ry 0 rz -180 deg; joints [-27.187, 50.674, -79.414, 30.362, 115.322, 14.066]
  MoveL 5070 to (234.45, 38.24, 78.65) mm, rotated rx -180 ry 0 rz -180 deg; joints [-27.187, 50.674, -79.414, 30.362, 115.322, 14.066]
  Call Extruder(203.07009)
  MoveL 5071 to (234.9, 38.57, 78.65) mm, rotated rx 180 ry 0 rz 180 deg; joints [-27.245, 50.731, -79.412, 30.41, 115.257, 14.06]
  MoveL 5072 to (234.9, 38.57, 78.65) mm, rotated rx 180 ry 0 rz 180 deg; joints [-27.245, 50.731, -79.412, 30.41, 115.257, 14.06]
  Call Extruder(203.40469)
  MoveL 5073 to (235.35, 38.9, 78.65) mm, rotated rx 180 ry 0 rz 180 deg; joints [-27.302, 50.788, -79.41, 30.458, 115.192, 14.053]
  Call Extruder(204.23264)
  MoveL 5074 to (236.39, 39.81, 78.65) mm, rotated rx -180 ry 0 rz 180 deg; joints [-27.525, 50.927, -79.405, 30.662, 115.015, 14.073]
  Call Extruder(205.06059)
  MoveL 5075 to (237.3, 40.85, 78.65) mm, rotated rx -180 ry 0 rz 180 deg; joints [-27.851, 51.059, -79.399, 30.978, 114.816, 14.142]
  Call Extruder(205.22789)
  MoveL 5076 to (237.47, 41.07, 78.65) mm, rotated rx -180 ry 0 rz 180 deg; joints [-27.932, 51.085, -79.398, 31.058, 114.773, 14.163]
  MoveL 5077 to (237.47, 41.07, 78.65) mm, rotated rx -180 ry 0 rz 180 deg; joints [-27.932, 51.085, -79.398, 31.058, 114.773, 14.163]
  Call Extruder(205.56130)
  MoveL 5078 to (237.79, 41.52, 78.65) mm, rotated rx 180 ry 0 rz -180 deg; joints [-28.091, 51.137, -79.395, 31.215, 114.688, 14.203]
  MoveL 5079 to (237.79, 41.52, 78.65) mm, rotated rx 180 ry 0 rz -180 deg; joints [-28.091, 51.137, -79.395, 31.215, 114.688, 14.203]
  Call Extruder(205.89353)
  MoveL 5080 to (238.12, 41.97, 78.65) mm, rotated rx -180 ry 0 rz 180 deg; joints [-28.249, 51.188, -79.393, 31.37, 114.603, 14.242]
  MoveL 5081 to (238.12, 41.97, 78.65) mm, rotated rx -180 ry 0 rz 180 deg; joints [-28.249, 51.188, -79.393, 31.37, 114.603, 14.242]
  Call Extruder(206.01123)
  MoveL 5082 to (238.22, 42.15, 78.65) mm, rotated rx -180 ry 0 rz 180 deg; joints [-28.315, 51.205, -79.392, 31.437, 114.571, 14.262]
  MoveL 5083 to (238.22, 42.15, 78.65) mm, rotated rx -180 ry 0 rz 180 deg; joints [-28.315, 51.205, -79.392, 31.437, 114.571, 14.262]
  Call Extruder(206.21895)
  MoveL 5084 to (238.4, 42.45, 78.65) mm, rotated rx -180 ry 0 rz 180 deg; joints [-28.434, 51.236, -79.39, 31.555, 114.515, 14.296]
  MoveL 5085 to (238.4, 42.45, 78.65) mm, rotated rx -180 ry 0 rz 180 deg; joints [-28.434, 51.236, -79.39, 31.555, 114.515, 14.296]
  Call Extruder(206.42590)
  MoveL 5086 to (238.57, 42.75, 78.65) mm, rotated rx -180 ry 0 rz 180 deg; joints [-28.552, 51.267, -79.389, 31.673, 114.458, 14.329]
  MoveL 5087 to (238.57, 42.75, 78.65) mm, rotated rx -180 ry 0 rz 180 deg; joints [-28.552, 51.267, -79.389, 31.673, 114.458, 14.329]
  Call Extruder(206.63206)
  MoveL 5088 to (238.75, 43.06, 78.65) mm, rotated rx -180 ry 0 rz -180 deg; joints [-28.669, 51.297, -79.387, 31.79, 114.402, 14.362]
  MoveL 5089 to (238.75, 43.06, 78.65) mm, rotated rx -180 ry 0 rz -180 deg; joints [-28.669, 51.297, -79.387, 31.79, 114.402, 14.362]
  Call Extruder(206.81375)
  MoveL 5090 to (238.89, 43.34, 78.65) mm, rotated rx 180 ry 0 rz 180 deg; joints [-28.78, 51.324, -79.386, 31.901, 114.35, 14.395]
  MoveL 5091 to (238.89, 43.34, 78.65) mm, rotated rx 180 ry 0 rz 180 deg; joints [-28.78, 51.324, -79.386, 31.901, 114.35, 14.395]
  Call Extruder(206.97176)
  MoveL 5092 to (239, 43.58, 78.65) mm, rotated rx 180 ry 0 rz 180 deg; joints [-28.886, 51.345, -79.384, 32.009, 114.304, 14.428]
  MoveL 5093 to (239, 43.58, 78.65) mm, rotated rx 180 ry 0 rz 180 deg; joints [-28.886, 51.345, -79.384, 32.009, 114.304, 14.428]
  Call Extruder(207.12917)
  MoveL 5094 to (239.11, 43.83, 78.65) mm, rotated rx 180 ry 0 rz 180 deg; joints [-28.991, 51.367, -79.383, 32.115, 114.259, 14.46]
  MoveL 5095 to (239.11, 43.83, 78.65) mm, rotated rx 180 ry 0 rz 180 deg; joints [-28.991, 51.367, -79.383, 32.115, 114.259, 14.46]
  Call Extruder(207.31188)
  MoveL 5096 to (239.22, 44.12, 78.65) mm, rotated rx -180 ry 0 rz 180 deg; joints [-29.116, 51.393, -79.382, 32.241, 114.205, 14.499]
  MoveL 5097 to (239.22, 44.12, 78.65) mm, rotated rx -180 ry 0 rz 180 deg; joints [-29.116, 51.393, -79.382, 32.241, 114.205, 14.499]
  Call Extruder(207.49384)
  MoveL 5098 to (239.35, 44.42, 78.65) mm, rotated rx 180 ry 0 rz 180 deg; joints [-29.24, 51.418, -79.38, 32.366, 114.151, 14.537]
  MoveL 5099 to (239.35, 44.42, 78.65) mm, rotated rx 180 ry 0 rz 180 deg; joints [-29.24, 51.418, -79.38, 32.366, 114.151, 14.537]
  Call Extruder(207.64117)
  MoveL 5100 to (239.44, 44.66, 78.65) mm, rotated rx -180 ry 0 rz 180 deg; joints [-29.343, 51.438, -79.379, 32.471, 114.107, 14.57]
  MoveL 5101 to (239.44, 44.66, 78.65) mm, rotated rx -180 ry 0 rz 180 deg; joints [-29.343, 51.438, -79.379, 32.471, 114.107, 14.57]
  Call Extruder(207.75441)
  MoveL 5102 to (239.5, 44.85, 78.65) mm, rotated rx -180 ry 0 rz 180 deg; joints [-29.428, 51.453, -79.378, 32.556, 114.073, 14.597]
  MoveL 5103 to (239.5, 44.85, 78.65) mm, rotated rx -180 ry 0 rz 180 deg; joints [-29.428, 51.453, -79.378, 32.556, 114.073, 14.597]
  Call Extruder(207.86720)
  MoveL 5104 to (239.56, 45.03, 78.65) mm, rotated rx -180 ry 0 rz 180 deg; joints [-29.512, 51.468, -79.377, 32.641, 114.038, 14.624]
  MoveL 5105 to (239.56, 45.03, 78.65) mm, rotated rx -180 ry 0 rz 180 deg; joints [-29.512, 51.468, -79.377, 32.641, 114.038, 14.624]
  Call Extruder(207.97954)
  MoveL 5106 to (239.62, 45.22, 78.65) mm, rotated rx -180 ry 0 rz 180 deg; joints [-29.596, 51.483, -79.376, 32.726, 114.004, 14.651]
  MoveL 5107 to (239.62, 45.22, 78.65) mm, rotated rx -180 ry 0 rz 180 deg; joints [-29.596, 51.483, -79.376, 32.726, 114.004, 14.651]
  Call Extruder(208.09145)
  MoveL 5108 to (239.68, 45.41, 78.65) mm, rotated rx 180 ry 0 rz 180 deg; joints [-29.679, 51.497, -79.375, 32.811, 113.969, 14.677]
  MoveL 5109 to (239.68, 45.41, 78.65) mm, rotated rx 180 ry 0 rz 180 deg; joints [-29.679, 51.497, -79.375, 32.811, 113.969, 14.677]
  Call Extruder(208.21285)
  MoveL 5110 to (239.75, 45.62, 78.65) mm, rotated rx -180 ry 0 rz 180 deg; joints [-29.77, 51.514, -79.374, 32.904, 113.932, 14.706]
  MoveL 5111 to (239.75, 45.62, 78.65) mm, rotated rx -180 ry 0 rz 180 deg; joints [-29.77, 51.514, -79.374, 32.904, 113.932, 14.706]
  Call Extruder(208.34364)
  MoveL 5112 to (239.82, 45.84, 78.65) mm, rotated rx -180 ry 0 rz 180 deg; joints [-29.871, 51.531, -79.373, 33.005, 113.891, 14.738]
  MoveL 5113 to (239.82, 45.84, 78.65) mm, rotated rx -180 ry 0 rz 180 deg; joints [-29.871, 51.531, -79.373, 33.005, 113.891, 14.738]
  Call Extruder(208.47386)
  MoveL 5114 to (239.88, 46.06, 78.65) mm, rotated rx 180 ry 0 rz -180 deg; joints [-29.97, 51.548, -79.372, 33.106, 113.85, 14.77]
  MoveL 5115 to (239.88, 46.06, 78.65) mm, rotated rx 180 ry 0 rz -180 deg; joints [-29.97, 51.548, -79.372, 33.106, 113.85, 14.77]
  Call Extruder(208.60352)
  MoveL 5116 to (239.95, 46.29, 78.65) mm, rotated rx -180 ry 0 rz 180 deg; joints [-30.069, 51.566, -79.371, 33.206, 113.809, 14.801]
  MoveL 5117 to (239.95, 46.29, 78.65) mm, rotated rx -180 ry 0 rz 180 deg; joints [-30.069, 51.566, -79.371, 33.206, 113.809, 14.801]
  Call Extruder(208.73262)
  MoveL 5118 to (240.02, 46.51, 78.65) mm, rotated rx 180 ry 0 rz 180 deg; joints [-30.168, 51.583, -79.37, 33.307, 113.768, 14.832]
  MoveL 5119 to (240.02, 46.51, 78.65) mm, rotated rx 180 ry 0 rz 180 deg; joints [-30.168, 51.583, -79.37, 33.307, 113.768, 14.832]
  Call Extruder(208.84768)
  MoveL 5120 to (240.06, 46.72, 78.65) mm, rotated rx -180 ry 0 rz 180 deg; joints [-30.263, 51.597, -79.369, 33.403, 113.731, 14.864]
  MoveL 5121 to (240.06, 46.72, 78.65) mm, rotated rx -180 ry 0 rz 180 deg; joints [-30.263, 51.597, -79.369, 33.403, 113.731, 14.864]
  Call Extruder(208.96228)
  MoveL 5122 to (240.11, 46.92, 78.65) mm, rotated rx -180 ry 0 rz 180 deg; joints [-30.358, 51.612, -79.368, 33.5, 113.694, 14.895]
  MoveL 5123 to (240.11, 46.92, 78.65) mm, rotated rx -180 ry 0 rz 180 deg; joints [-30.358, 51.612, -79.368, 33.5, 113.694, 14.895]
  Call Extruder(209.07643)
  MoveL 5124 to (240.15, 47.12, 78.65) mm, rotated rx -180 ry 0 rz -180 deg; joints [-30.453, 51.626, -79.367, 33.596, 113.657, 14.925]
  MoveL 5125 to (240.15, 47.12, 78.65) mm, rotated rx -180 ry 0 rz -180 deg; joints [-30.453, 51.626, -79.367, 33.596, 113.657, 14.925]
  Call Extruder(209.19012)
  MoveL 5126 to (240.2, 47.33, 78.65) mm, rotated rx -180 ry 0 rz 180 deg; joints [-30.548, 51.64, -79.366, 33.692, 113.62, 14.956]
  MoveL 5127 to (240.2, 47.33, 78.65) mm, rotated rx -180 ry 0 rz 180 deg; joints [-30.548, 51.64, -79.366, 33.692, 113.62, 14.956]
  Call Extruder(209.31554)
  MoveL 5128 to (240.24, 47.56, 78.65) mm, rotated rx -180 ry 0 rz 180 deg; joints [-30.653, 51.656, -79.365, 33.798, 113.579, 14.99]
  MoveL 5129 to (240.24, 47.56, 78.65) mm, rotated rx -180 ry 0 rz 180 deg; joints [-30.653, 51.656, -79.365, 33.798, 113.579, 14.99]
  Call Extruder(209.45251)
  MoveL 5130 to (240.29, 47.8, 78.65) mm, rotated rx 180 ry 0 rz 180 deg; joints [-30.768, 51.674, -79.364, 33.916, 113.533, 15.028]
  MoveL 5131 to (240.29, 47.8, 78.65) mm, rotated rx 180 ry 0 rz 180 deg; joints [-30.768, 51.674, -79.364, 33.916, 113.533, 15.028]
  Call Extruder(209.58888)
  MoveL 5132 to (240.34, 48.05, 78.65) mm, rotated rx -180 ry 0 rz -180 deg; joints [-30.884, 51.691, -79.363, 34.033, 113.488, 15.065]
  MoveL 5133 to (240.34, 48.05, 78.65) mm, rotated rx -180 ry 0 rz -180 deg; joints [-30.884, 51.691, -79.363, 34.033, 113.488, 15.065]
  Call Extruder(209.72464)
  MoveL 5134 to (240.39, 48.3, 78.65) mm, rotated rx -180 ry 0 rz 180 deg; joints [-30.999, 51.708, -79.361, 34.15, 113.443, 15.102]
  MoveL 5135 to (240.39, 48.3, 78.65) mm, rotated rx -180 ry 0 rz 180 deg; joints [-30.999, 51.708, -79.361, 34.15, 113.443, 15.102]
  Call Extruder(209.85978)
  MoveL 5136 to (240.44, 48.55, 78.65) mm, rotated rx 180 ry 0 rz -180 deg; joints [-31.114, 51.725, -79.36, 34.266, 113.397, 15.139]
  MoveL 5137 to (240.44, 48.55, 78.65) mm, rotated rx 180 ry 0 rz -180 deg; joints [-31.114, 51.725, -79.36, 34.266, 113.397, 15.139]
  Call Extruder(209.99432)
  MoveL 5138 to (240.49, 48.8, 78.65) mm, rotated rx -180 ry 0 rz 180 deg; joints [-31.228, 51.743, -79.359, 34.382, 113.352, 15.175]
  MoveL 5139 to (240.49, 48.8, 78.65) mm, rotated rx -180 ry 0 rz 180 deg; joints [-31.228, 51.743, -79.359, 34.382, 113.352, 15.175]
  Call Extruder(210.12825)
  MoveL 5140 to (240.54, 49.05, 78.65) mm, rotated rx -180 ry 0 rz 180 deg; joints [-31.342, 51.76, -79.358, 34.497, 113.307, 15.211]
  MoveL 5141 to (240.54, 49.05, 78.65) mm, rotated rx -180 ry 0 rz 180 deg; joints [-31.342, 51.76, -79.358, 34.497, 113.307, 15.211]
  Call Extruder(210.27611)
  MoveL 5142 to (240.59, 49.33, 78.65) mm, rotated rx -180 ry 0 rz 180 deg; joints [-31.47, 51.779, -79.356, 34.626, 113.257, 15.252]
  MoveL 5143 to (240.59, 49.33, 78.65) mm, rotated rx -180 ry 0 rz 180 deg; joints [-31.47, 51.779, -79.356, 34.626, 113.257, 15.252]
  Call Extruder(210.43786)
  MoveL 5144 to (240.64, 49.63, 78.65) mm, rotated rx -180 ry 0 rz 180 deg; joints [-31.612, 51.799, -79.355, 34.771, 113.201, 15.297]
  MoveL 5145 to (240.64, 49.63, 78.65) mm, rotated rx -180 ry 0 rz 180 deg; joints [-31.612, 51.799, -79.355, 34.771, 113.201, 15.297]
  Call Extruder(210.59887)
  MoveL 5146 to (240.69, 49.94, 78.65) mm, rotated rx 180 ry 0 rz 180 deg; joints [-31.755, 51.82, -79.353, 34.914, 113.146, 15.342]
  MoveL 5147 to (240.69, 49.94, 78.65) mm, rotated rx 180 ry 0 rz 180 deg; joints [-31.755, 51.82, -79.353, 34.914, 113.146, 15.342]
  Call Extruder(210.75916)
  MoveL 5148 to (240.73, 50.24, 78.65) mm, rotated rx -180 ry 0 rz 180 deg; joints [-31.895, 51.84, -79.352, 35.057, 113.09, 15.386]
  MoveL 5149 to (240.73, 50.24, 78.65) mm, rotated rx -180 ry 0 rz 180 deg; joints [-31.895, 51.84, -79.352, 35.057, 113.09, 15.386]
  Call Extruder(210.91872)
  MoveL 5150 to (240.78, 50.55, 78.65) mm, rotated rx -180 ry 0 rz 180 deg; joints [-32.036, 51.861, -79.35, 35.199, 113.035, 15.43]
  MoveL 5151 to (240.78, 50.55, 78.65) mm, rotated rx -180 ry 0 rz 180 deg; joints [-32.036, 51.861, -79.35, 35.199, 113.035, 15.43]
  Call Extruder(211.07756)
  MoveL 5152 to (240.83, 50.86, 78.65) mm, rotated rx -180 ry 0 rz 180 deg; joints [-32.176, 51.881, -79.349, 35.34, 112.98, 15.474]
  MoveL 5153 to (240.83, 50.86, 78.65) mm, rotated rx -180 ry 0 rz 180 deg; joints [-32.176, 51.881, -79.349, 35.34, 112.98, 15.474]
  Call Extruder(211.25623)
  MoveL 5154 to (240.88, 51.2, 78.65) mm, rotated rx -180 ry 0 rz 180 deg; joints [-32.337, 51.904, -79.347, 35.502, 112.917, 15.524]
  MoveL 5155 to (240.88, 51.2, 78.65) mm, rotated rx -180 ry 0 rz 180 deg; joints [-32.337, 51.904, -79.347, 35.502, 112.917, 15.524]
  Call Extruder(211.45467)
  MoveL 5156 to (240.93, 51.59, 78.65) mm, rotated rx 180 ry 0 rz 180 deg; joints [-32.518, 51.929, -79.345, 35.685, 112.846, 15.58]
  MoveL 5157 to (240.93, 51.59, 78.65) mm, rotated rx 180 ry 0 rz 180 deg; joints [-32.518, 51.929, -79.345, 35.685, 112.846, 15.58]
  Call Extruder(211.65225)
  MoveL 5158 to (240.97, 51.98, 78.65) mm, rotated rx -180 ry 0 rz 180 deg; joints [-32.697, 51.954, -79.343, 35.866, 112.776, 15.636]
  MoveL 5159 to (240.97, 51.98, 78.65) mm, rotated rx -180 ry 0 rz 180 deg; joints [-32.697, 51.954, -79.343, 35.866, 112.776, 15.636]
  Call Extruder(211.84895)
  MoveL 5160 to (241.02, 52.36, 78.65) mm, rotated rx -180 ry 0 rz 180 deg; joints [-32.876, 51.979, -79.341, 36.046, 112.706, 15.691]
  MoveL 5161 to (241.02, 52.36, 78.65) mm, rotated rx -180 ry 0 rz 180 deg; joints [-32.876, 51.979, -79.341, 36.046, 112.706, 15.691]
  Call Extruder(212.04479)
  MoveL 5162 to (241.06, 52.75, 78.65) mm, rotated rx 180 ry 0 rz 180 deg; joints [-33.055, 52.004, -79.339, 36.225, 112.636, 15.745]
  MoveL 5163 to (241.06, 52.75, 78.65) mm, rotated rx 180 ry 0 rz 180 deg; joints [-33.055, 52.004, -79.339, 36.225, 112.636, 15.745]
  Call Extruder(212.34023)
  MoveL 5164 to (241.11, 53.34, 78.65) mm, rotated rx 180 ry 0 rz 180 deg; joints [-33.331, 52.04, -79.336, 36.504, 112.529, 15.831]
  MoveL 5165 to (241.11, 53.34, 78.65) mm, rotated rx 180 ry 0 rz 180 deg; joints [-33.331, 52.04, -79.336, 36.504, 112.529, 15.831]
  Call Extruder(212.63433)
  MoveL 5166 to (241.16, 53.93, 78.65) mm, rotated rx 180 ry 0 rz 180 deg; joints [-33.606, 52.077, -79.333, 36.78, 112.422, 15.915]
  MoveL 5167 to (241.16, 53.93, 78.65) mm, rotated rx 180 ry 0 rz 180 deg; joints [-33.606, 52.077, -79.333, 36.78, 112.422, 15.915]
  Call Extruder(212.92711)
  MoveL 5168 to (241.2, 54.52, 78.65) mm, rotated rx -180 ry 0 rz -180 deg; joints [-33.878, 52.114, -79.33, 37.053, 112.315, 15.996]
  MoveL 5169 to (241.2, 54.52, 78.65) mm, rotated rx -180 ry 0 rz -180 deg; joints [-33.878, 52.114, -79.33, 37.053, 112.315, 15.996]
  Call Extruder(213.50056)
  MoveL 5170 to (241.25, 55.68, 78.65) mm, rotated rx -180 ry 0 rz 180 deg; joints [-34.425, 52.183, -79.324, 37.602, 112.104, 16.161]
  MoveL 5171 to (241.25, 55.68, 78.65) mm, rotated rx -180 ry 0 rz 180 deg; joints [-34.425, 52.183, -79.324, 37.602, 112.104, 16.161]
  Call Extruder(214.21439)
  MoveL 5172 to (241.29, 57.14, 78.65) mm, rotated rx -180 ry 0 rz 180 deg; joints [-35.104, 52.269, -79.316, 38.282, 111.839, 16.362]
  Call Extruder(256.27928)
  MoveL 5173 to (241.29, 142.86, 78.65) mm, rotated rx -180 ry 0 rz 180 deg; joints [-60.361, 58.255, -77.917, 61.817, 99.579, 17.253]
  Call Extruder(256.70771)
  MoveL 5174 to (241.27, 143.74, 78.65) mm, rotated rx -180 ry 0 rz 180 deg; joints [-60.516, 58.317, -77.891, 61.954, 99.491, 17.199]
  MoveL 5175 to (241.27, 143.74, 78.65) mm, rotated rx -180 ry 0 rz 180 deg; joints [-60.516, 58.317, -77.891, 61.954, 99.491, 17.199]
  Call Extruder(257.28116)
  MoveL 5176 to (241.22, 144.9, 78.65) mm, rotated rx -180 ry 0 rz 180 deg; joints [-60.726, 58.4, -77.857, 62.141, 99.374, 17.128]
  MoveL 5177 to (241.22, 144.9, 78.65) mm, rotated rx -180 ry 0 rz 180 deg; joints [-60.726, 58.4, -77.857, 62.141, 99.374, 17.128]
  Call Extruder(257.71549)
  MoveL 5178 to (241.18, 145.77, 78.65) mm, rotated rx 180 ry 0 rz -180 deg; joints [-60.887, 58.461, -77.832, 62.284, 99.286, 17.075]
  MoveL 5179 to (241.18, 145.77, 78.65) mm, rotated rx 180 ry 0 rz -180 deg; joints [-60.887, 58.461, -77.832, 62.284, 99.286, 17.075]
  Call Extruder(258.00960)
  MoveL 5180 to (241.13, 146.36, 78.65) mm, rotated rx 180 ry 0 rz -180 deg; joints [-61, 58.502, -77.815, 62.385, 99.226, 17.04]
  MoveL 5181 to (241.13, 146.36, 78.65) mm, rotated rx 180 ry 0 rz -180 deg; joints [-61, 58.502, -77.815, 62.385, 99.226, 17.04]
  Call Extruder(258.30504)
  MoveL 5182 to (241.09, 146.95, 78.65) mm, rotated rx 180 ry 0 rz 180 deg; joints [-61.111, 58.543, -77.797, 62.484, 99.167, 17.005]
  MoveL 5183 to (241.09, 146.95, 78.65) mm, rotated rx 180 ry 0 rz 180 deg; joints [-61.111, 58.543, -77.797, 62.484, 99.167, 17.005]
  Call Extruder(258.55130)
  MoveL 5184 to (241.04, 147.44, 78.65) mm, rotated rx 180 ry 0 rz 180 deg; joints [-61.205, 58.577, -77.783, 62.568, 99.117, 16.977]
  MoveL 5185 to (241.04, 147.44, 78.65) mm, rotated rx 180 ry 0 rz 180 deg; joints [-61.205, 58.577, -77.783, 62.568, 99.117, 16.977]
  Call Extruder(258.74800)
  MoveL 5186 to (240.99, 147.83, 78.65) mm, rotated rx -180 ry 0 rz 180 deg; joints [-61.282, 58.603, -77.772, 62.638, 99.078, 16.955]
  MoveL 5187 to (240.99, 147.83, 78.65) mm, rotated rx -180 ry 0 rz 180 deg; joints [-61.282, 58.603, -77.772, 62.638, 99.078, 16.955]
  Call Extruder(258.94558)
  MoveL 5188 to (240.95, 148.22, 78.65) mm, rotated rx -180 ry 0 rz 180 deg; joints [-61.359, 58.629, -77.76, 62.707, 99.038, 16.933]
  MoveL 5189 to (240.95, 148.22, 78.65) mm, rotated rx -180 ry 0 rz 180 deg; joints [-61.359, 58.629, -77.76, 62.707, 99.038, 16.933]
  Call Extruder(259.14402)
  MoveL 5190 to (240.9, 148.6, 78.65) mm, rotated rx 180 ry 0 rz 180 deg; joints [-61.436, 58.655, -77.749, 62.776, 98.999, 16.911]
  MoveL 5191 to (240.9, 148.6, 78.65) mm, rotated rx 180 ry 0 rz 180 deg; joints [-61.436, 58.655, -77.749, 62.776, 98.999, 16.911]
  Call Extruder(259.34333)
  MoveL 5192 to (240.86, 148.99, 78.65) mm, rotated rx 180 ry 0 rz -180 deg; joints [-61.512, 58.681, -77.738, 62.844, 98.959, 16.888]
  MoveL 5193 to (240.86, 148.99, 78.65) mm, rotated rx 180 ry 0 rz -180 deg; joints [-61.512, 58.681, -77.738, 62.844, 98.959, 16.888]
  Call Extruder(259.50216)
  MoveL 5194 to (240.81, 149.3, 78.65) mm, rotated rx 180 ry 0 rz 180 deg; joints [-61.575, 58.702, -77.729, 62.902, 98.928, 16.872]
  MoveL 5195 to (240.81, 149.3, 78.65) mm, rotated rx 180 ry 0 rz 180 deg; joints [-61.575, 58.702, -77.729, 62.902, 98.928, 16.872]
  Call Extruder(259.66172)
  MoveL 5196 to (240.76, 149.6, 78.65) mm, rotated rx -180 ry 0 rz -180 deg; joints [-61.639, 58.722, -77.72, 62.959, 98.896, 16.855]
  MoveL 5197 to (240.76, 149.6, 78.65) mm, rotated rx -180 ry 0 rz -180 deg; joints [-61.639, 58.722, -77.72, 62.959, 98.896, 16.855]
  Call Extruder(259.82201)
  MoveL 5198 to (240.71, 149.91, 78.65) mm, rotated rx 180 ry 0 rz 180 deg; joints [-61.702, 58.742, -77.711, 63.016, 98.864, 16.838]
  MoveL 5199 to (240.71, 149.91, 78.65) mm, rotated rx 180 ry 0 rz 180 deg; joints [-61.702, 58.742, -77.711, 63.016, 98.864, 16.838]
  Call Extruder(259.98302)
  MoveL 5200 to (240.66, 150.21, 78.65) mm, rotated rx 180 ry 0 rz 180 deg; joints [-61.765, 58.762, -77.702, 63.074, 98.833, 16.822]
  MoveL 5201 to (240.66, 150.21, 78.65) mm, rotated rx 180 ry 0 rz 180 deg; joints [-61.765, 58.762, -77.702, 63.074, 98.833, 16.822]
  Call Extruder(260.14477)
  MoveL 5202 to (240.61, 150.52, 78.65) mm, rotated rx -180 ry 0 rz 180 deg; joints [-61.828, 58.782, -77.693, 63.13, 98.802, 16.805]
  MoveL 5203 to (240.61, 150.52, 78.65) mm, rotated rx -180 ry 0 rz 180 deg; joints [-61.828, 58.782, -77.693, 63.13, 98.802, 16.805]
  Call Extruder(260.30724)
  MoveL 5204 to (240.56, 150.83, 78.65) mm, rotated rx -180 ry 0 rz 180 deg; joints [-61.891, 58.803, -77.684, 63.187, 98.77, 16.788]
  MoveL 5205 to (240.56, 150.83, 78.65) mm, rotated rx -180 ry 0 rz 180 deg; joints [-61.891, 58.803, -77.684, 63.187, 98.77, 16.788]
  Call Extruder(260.44117)
  MoveL 5206 to (240.52, 151.07, 78.65) mm, rotated rx 180 ry 0 rz 180 deg; joints [-61.944, 58.819, -77.677, 63.236, 98.744, 16.775]
  MoveL 5207 to (240.52, 151.07, 78.65) mm, rotated rx 180 ry 0 rz 180 deg; joints [-61.944, 58.819, -77.677, 63.236, 98.744, 16.775]
  Call Extruder(260.57570)
  MoveL 5208 to (240.47, 151.32, 78.65) mm, rotated rx 180 ry 0 rz -180 deg; joints [-61.998, 58.835, -77.67, 63.285, 98.718, 16.761]
  MoveL 5209 to (240.47, 151.32, 78.65) mm, rotated rx 180 ry 0 rz -180 deg; joints [-61.998, 58.835, -77.67, 63.285, 98.718, 16.761]
  Call Extruder(260.71085)
  MoveL 5210 to (240.42, 151.57, 78.65) mm, rotated rx 180 ry 0 rz 180 deg; joints [-62.052, 58.851, -77.663, 63.334, 98.692, 16.748]
  MoveL 5211 to (240.42, 151.57, 78.65) mm, rotated rx 180 ry 0 rz 180 deg; joints [-62.052, 58.851, -77.663, 63.334, 98.692, 16.748]
  Call Extruder(260.84661)
  MoveL 5212 to (240.37, 151.82, 78.65) mm, rotated rx -180 ry 0 rz 180 deg; joints [-62.105, 58.867, -77.656, 63.383, 98.667, 16.735]
  MoveL 5213 to (240.37, 151.82, 78.65) mm, rotated rx -180 ry 0 rz 180 deg; joints [-62.105, 58.867, -77.656, 63.383, 98.667, 16.735]
  Call Extruder(260.98297)
  MoveL 5214 to (240.32, 152.07, 78.65) mm, rotated rx 180 ry 0 rz 180 deg; joints [-62.159, 58.883, -77.649, 63.431, 98.641, 16.722]
  MoveL 5215 to (240.32, 152.07, 78.65) mm, rotated rx 180 ry 0 rz 180 deg; joints [-62.159, 58.883, -77.649, 63.431, 98.641, 16.722]
  Call Extruder(261.11995)
  MoveL 5216 to (240.27, 152.32, 78.65) mm, rotated rx 180 ry 0 rz -180 deg; joints [-62.212, 58.899, -77.641, 63.48, 98.615, 16.708]
  MoveL 5217 to (240.27, 152.32, 78.65) mm, rotated rx 180 ry 0 rz -180 deg; joints [-62.212, 58.899, -77.641, 63.48, 98.615, 16.708]
  Call Extruder(261.25754)
  MoveL 5218 to (240.22, 152.57, 78.65) mm, rotated rx -180 ry 0 rz 180 deg; joints [-62.265, 58.915, -77.634, 63.528, 98.589, 16.695]
  MoveL 5219 to (240.22, 152.57, 78.65) mm, rotated rx -180 ry 0 rz 180 deg; joints [-62.265, 58.915, -77.634, 63.528, 98.589, 16.695]
  Call Extruder(261.37124)
  MoveL 5220 to (240.17, 152.77, 78.65) mm, rotated rx -180 ry 0 rz 180 deg; joints [-62.31, 58.928, -77.628, 63.569, 98.568, 16.684]
  MoveL 5221 to (240.17, 152.77, 78.65) mm, rotated rx -180 ry 0 rz 180 deg; joints [-62.31, 58.928, -77.628, 63.569, 98.568, 16.684]
  Call Extruder(261.48539)
  MoveL 5222 to (240.13, 152.98, 78.65) mm, rotated rx -180 ry 0 rz 180 deg; joints [-62.355, 58.941, -77.622, 63.609, 98.547, 16.674]
  MoveL 5223 to (240.13, 152.98, 78.65) mm, rotated rx -180 ry 0 rz 180 deg; joints [-62.355, 58.941, -77.622, 63.609, 98.547, 16.674]
  Call Extruder(261.59999)
  MoveL 5224 to (240.08, 153.18, 78.65) mm, rotated rx 180 ry 0 rz 180 deg; joints [-62.399, 58.954, -77.616, 63.65, 98.526, 16.663]
  MoveL 5225 to (240.08, 153.18, 78.65) mm, rotated rx 180 ry 0 rz 180 deg; joints [-62.399, 58.954, -77.616, 63.65, 98.526, 16.663]
  Call Extruder(261.71505)
  MoveL 5226 to (240.04, 153.39, 78.65) mm, rotated rx -180 ry 0 rz -180 deg; joints [-62.444, 58.967, -77.61, 63.69, 98.505, 16.652]
  MoveL 5227 to (240.04, 153.39, 78.65) mm, rotated rx -180 ry 0 rz -180 deg; joints [-62.444, 58.967, -77.61, 63.69, 98.505, 16.652]
  Call Extruder(261.83727)
  MoveL 5228 to (239.98, 153.6, 78.65) mm, rotated rx -180 ry 0 rz 180 deg; joints [-62.493, 58.981, -77.604, 63.735, 98.482, 16.641]
  MoveL 5229 to (239.98, 153.6, 78.65) mm, rotated rx -180 ry 0 rz 180 deg; joints [-62.493, 58.981, -77.604, 63.735, 98.482, 16.641]
  Call Extruder(261.96693)
  MoveL 5230 to (239.92, 153.82, 78.65) mm, rotated rx -180 ry 0 rz 180 deg; joints [-62.547, 58.994, -77.598, 63.785, 98.458, 16.631]
  MoveL 5231 to (239.92, 153.82, 78.65) mm, rotated rx -180 ry 0 rz 180 deg; joints [-62.547, 58.994, -77.598, 63.785, 98.458, 16.631]
  Call Extruder(262.09716)
  MoveL 5232 to (239.85, 154.05, 78.65) mm, rotated rx -180 ry 0 rz 180 deg; joints [-62.601, 59.008, -77.592, 63.835, 98.434, 16.621]
  MoveL 5233 to (239.85, 154.05, 78.65) mm, rotated rx -180 ry 0 rz 180 deg; joints [-62.601, 59.008, -77.592, 63.835, 98.434, 16.621]
  Call Extruder(262.22795)
  MoveL 5234 to (239.78, 154.27, 78.65) mm, rotated rx 180 ry 0 rz -180 deg; joints [-62.654, 59.021, -77.586, 63.884, 98.409, 16.611]
  MoveL 5235 to (239.78, 154.27, 78.65) mm, rotated rx 180 ry 0 rz -180 deg; joints [-62.654, 59.021, -77.586, 63.884, 98.409, 16.611]
  Call Extruder(262.35930)
  MoveL 5236 to (239.71, 154.5, 78.65) mm, rotated rx 180 ry 0 rz 180 deg; joints [-62.708, 59.035, -77.579, 63.934, 98.385, 16.6]
  MoveL 5237 to (239.71, 154.5, 78.65) mm, rotated rx 180 ry 0 rz 180 deg; joints [-62.708, 59.035, -77.579, 63.934, 98.385, 16.6]
  Call Extruder(262.47120)
  MoveL 5238 to (239.65, 154.68, 78.65) mm, rotated rx 180 ry 0 rz 180 deg; joints [-62.754, 59.046, -77.574, 63.976, 98.365, 16.592]
  MoveL 5239 to (239.65, 154.68, 78.65) mm, rotated rx 180 ry 0 rz 180 deg; joints [-62.754, 59.046, -77.574, 63.976, 98.365, 16.592]
  Call Extruder(262.58355)
  MoveL 5240 to (239.59, 154.87, 78.65) mm, rotated rx -180 ry 0 rz 180 deg; joints [-62.801, 59.058, -77.569, 64.019, 98.344, 16.583]
  MoveL 5241 to (239.59, 154.87, 78.65) mm, rotated rx -180 ry 0 rz 180 deg; joints [-62.801, 59.058, -77.569, 64.019, 98.344, 16.583]
  Call Extruder(262.69634)
  MoveL 5242 to (239.53, 155.06, 78.65) mm, rotated rx 180 ry 0 rz -180 deg; joints [-62.847, 59.069, -77.564, 64.062, 98.324, 16.575]
  MoveL 5243 to (239.53, 155.06, 78.65) mm, rotated rx 180 ry 0 rz -180 deg; joints [-62.847, 59.069, -77.564, 64.062, 98.324, 16.575]
  Call Extruder(262.80957)
  MoveL 5244 to (239.47, 155.25, 78.65) mm, rotated rx 180 ry 0 rz -180 deg; joints [-62.893, 59.08, -77.558, 64.104, 98.303, 16.566]
  MoveL 5245 to (239.47, 155.25, 78.65) mm, rotated rx 180 ry 0 rz -180 deg; joints [-62.893, 59.08, -77.558, 64.104, 98.303, 16.566]
  Call Extruder(262.92325)
  MoveL 5246 to (239.41, 155.44, 78.65) mm, rotated rx -180 ry 0 rz -180 deg; joints [-62.939, 59.091, -77.553, 64.146, 98.283, 16.557]
  MoveL 5247 to (239.41, 155.44, 78.65) mm, rotated rx -180 ry 0 rz -180 deg; joints [-62.939, 59.091, -77.553, 64.146, 98.283, 16.557]
  Call Extruder(263.10521)
  MoveL 5248 to (239.29, 155.73, 78.65) mm, rotated rx -180 ry 0 rz -180 deg; joints [-63.018, 59.108, -77.545, 64.22, 98.25, 16.546]
  MoveL 5249 to (239.29, 155.73, 78.65) mm, rotated rx -180 ry 0 rz -180 deg; joints [-63.018, 59.108, -77.545, 64.22, 98.25, 16.546]
  Call Extruder(263.28793)
  MoveL 5250 to (239.17, 156.02, 78.65) mm, rotated rx -180 ry 0 rz 180 deg; joints [-63.097, 59.125, -77.538, 64.293, 98.217, 16.535]
  MoveL 5251 to (239.17, 156.02, 78.65) mm, rotated rx -180 ry 0 rz 180 deg; joints [-63.097, 59.125, -77.538, 64.293, 98.217, 16.535]
  Call Extruder(263.45835)
  MoveL 5252 to (239.05, 156.29, 78.65) mm, rotated rx -180 ry 0 rz 180 deg; joints [-63.17, 59.14, -77.53, 64.361, 98.187, 16.525]
  MoveL 5253 to (239.05, 156.29, 78.65) mm, rotated rx -180 ry 0 rz 180 deg; joints [-63.17, 59.14, -77.53, 64.361, 98.187, 16.525]
  Call Extruder(263.61637)
  MoveL 5254 to (238.94, 156.54, 78.65) mm, rotated rx 180 ry 0 rz -180 deg; joints [-63.238, 59.154, -77.524, 64.424, 98.158, 16.515]
  MoveL 5255 to (238.94, 156.54, 78.65) mm, rotated rx 180 ry 0 rz -180 deg; joints [-63.238, 59.154, -77.524, 64.424, 98.158, 16.515]
  Call Extruder(263.77499)
  MoveL 5256 to (238.84, 156.79, 78.65) mm, rotated rx -180 ry 0 rz 180 deg; joints [-63.306, 59.168, -77.517, 64.487, 98.13, 16.506]
  MoveL 5257 to (238.84, 156.79, 78.65) mm, rotated rx -180 ry 0 rz 180 deg; joints [-63.306, 59.168, -77.517, 64.487, 98.13, 16.506]
  Call Extruder(264.00155)
  MoveL 5258 to (238.65, 157.13, 78.65) mm, rotated rx -180 ry 0 rz 180 deg; joints [-63.41, 59.185, -77.509, 64.585, 98.089, 16.497]
  MoveL 5259 to (238.65, 157.13, 78.65) mm, rotated rx -180 ry 0 rz 180 deg; joints [-63.41, 59.185, -77.509, 64.585, 98.089, 16.497]
  Call Extruder(264.22896)
  MoveL 5260 to (238.46, 157.46, 78.65) mm, rotated rx 180 ry 0 rz -180 deg; joints [-63.514, 59.203, -77.501, 64.682, 98.049, 16.487]
  MoveL 5261 to (238.46, 157.46, 78.65) mm, rotated rx 180 ry 0 rz -180 deg; joints [-63.514, 59.203, -77.501, 64.682, 98.049, 16.487]
  Call Extruder(264.41617)
  MoveL 5262 to (238.3, 157.73, 78.65) mm, rotated rx -180 ry 0 rz -180 deg; joints [-63.601, 59.217, -77.494, 64.764, 98.016, 16.481]
  MoveL 5263 to (238.3, 157.73, 78.65) mm, rotated rx -180 ry 0 rz -180 deg; joints [-63.601, 59.217, -77.494, 64.764, 98.016, 16.481]
  Call Extruder(264.60408)
  MoveL 5264 to (238.13, 158.01, 78.65) mm, rotated rx 180 ry 0 rz 180 deg; joints [-63.687, 59.23, -77.488, 64.845, 97.982, 16.474]
  MoveL 5265 to (238.13, 158.01, 78.65) mm, rotated rx 180 ry 0 rz 180 deg; joints [-63.687, 59.23, -77.488, 64.845, 97.982, 16.474]
  Call Extruder(264.78361)
  MoveL 5266 to (237.96, 158.25, 78.65) mm, rotated rx 180 ry 0 rz -180 deg; joints [-63.774, 59.242, -77.482, 64.926, 97.951, 16.47]
  MoveL 5267 to (237.96, 158.25, 78.65) mm, rotated rx 180 ry 0 rz -180 deg; joints [-63.774, 59.242, -77.482, 64.926, 97.951, 16.47]
  Call Extruder(265.11703)
  MoveL 5268 to (237.63, 158.7, 78.65) mm, rotated rx 180 ry 0 rz 180 deg; joints [-63.934, 59.263, -77.472, 65.077, 97.892, 16.463]
  MoveL 5269 to (237.63, 158.7, 78.65) mm, rotated rx 180 ry 0 rz 180 deg; joints [-63.934, 59.263, -77.472, 65.077, 97.892, 16.463]
  Call Extruder(265.45163)
  MoveL 5270 to (237.3, 159.15, 78.65) mm, rotated rx 180 ry 0 rz 180 deg; joints [-64.094, 59.284, -77.462, 65.228, 97.834, 16.455]
  Call Extruder(266.27957)
  MoveL 5271 to (236.39, 160.19, 78.65) mm, rotated rx -180 ry 0 rz 180 deg; joints [-64.505, 59.327, -77.441, 65.618, 97.691, 16.45]
  Call Extruder(267.10752)
  MoveL 5272 to (235.35, 161.1, 78.65) mm, rotated rx 180 ry 0 rz -180 deg; joints [-64.933, 59.357, -77.426, 66.027, 97.551, 16.464]
  Call Extruder(267.27483)
  MoveL 5273 to (235.13, 161.27, 78.65) mm, rotated rx -180 ry 0 rz 180 deg; joints [-65.021, 59.362, -77.424, 66.111, 97.524, 16.469]
  MoveL 5274 to (235.13, 161.27, 78.65) mm, rotated rx -180 ry 0 rz 180 deg; joints [-65.021, 59.362, -77.424, 66.111, 97.524, 16.469]
  Call Extruder(267.60825)
  MoveL 5275 to (234.68, 161.59, 78.65) mm, rotated rx -180 ry 0 rz 180 deg; joints [-65.197, 59.37, -77.42, 66.28, 97.468, 16.479]
  MoveL 5276 to (234.68, 161.59, 78.65) mm, rotated rx -180 ry 0 rz 180 deg; joints [-65.197, 59.37, -77.42, 66.28, 97.468, 16.479]
  Call Extruder(267.94049)
  MoveL 5277 to (234.22, 161.92, 78.65) mm, rotated rx 180 ry 0 rz 180 deg; joints [-65.374, 59.379, -77.416, 66.449, 97.413, 16.489]
  MoveL 5278 to (234.22, 161.92, 78.65) mm, rotated rx 180 ry 0 rz 180 deg; joints [-65.374, 59.379, -77.416, 66.449, 97.413, 16.489]
  Call Extruder(268.05815)
  MoveL 5279 to (234.05, 162.02, 78.65) mm, rotated rx -180 ry 0 rz 180 deg; joints [-65.437, 59.38, -77.415, 66.51, 97.394, 16.495]
  MoveL 5280 to (234.05, 162.02, 78.65) mm, rotated rx -180 ry 0 rz 180 deg; joints [-65.437, 59.38, -77.415, 66.51, 97.394, 16.495]
  Call Extruder(268.26588)
  MoveL 5281 to (233.75, 162.2, 78.65) mm, rotated rx -180 ry 0 rz 180 deg; joints [-65.549, 59.383, -77.414, 66.618, 97.361, 16.505]
  MoveL 5282 to (233.75, 162.2, 78.65) mm, rotated rx -180 ry 0 rz 180 deg; joints [-65.549, 59.383, -77.414, 66.618, 97.361, 16.505]
  Call Extruder(268.47282)
  MoveL 5283 to (233.45, 162.37, 78.65) mm, rotated rx 180 ry 0 rz -180 deg; joints [-65.662, 59.386, -77.412, 66.726, 97.327, 16.516]
  MoveL 5284 to (233.45, 162.37, 78.65) mm, rotated rx 180 ry 0 rz -180 deg; joints [-65.662, 59.386, -77.412, 66.726, 97.327, 16.516]
  Call Extruder(268.67899)
  MoveL 5285 to (233.14, 162.55, 78.65) mm, rotated rx 180 ry 0 rz 180 deg; joints [-65.774, 59.389, -77.411, 66.834, 97.294, 16.526]
  MoveL 5286 to (233.14, 162.55, 78.65) mm, rotated rx 180 ry 0 rz 180 deg; joints [-65.774, 59.389, -77.411, 66.834, 97.294, 16.526]
  Call Extruder(268.86066)
  MoveL 5287 to (232.87, 162.69, 78.65) mm, rotated rx 180 ry 0 rz 180 deg; joints [-65.874, 59.39, -77.411, 66.931, 97.265, 16.536]
  MoveL 5288 to (232.87, 162.69, 78.65) mm, rotated rx 180 ry 0 rz 180 deg; joints [-65.874, 59.39, -77.411, 66.931, 97.265, 16.536]
  Call Extruder(269.01864)
  MoveL 5289 to (232.62, 162.8, 78.65) mm, rotated rx 180 ry 0 rz 180 deg; joints [-65.961, 59.39, -77.411, 67.015, 97.24, 16.547]
  MoveL 5290 to (232.62, 162.8, 78.65) mm, rotated rx 180 ry 0 rz 180 deg; joints [-65.961, 59.39, -77.411, 67.015, 97.24, 16.547]
  Call Extruder(269.17601)
  MoveL 5291 to (232.37, 162.9, 78.65) mm, rotated rx 180 ry 0 rz 180 deg; joints [-66.048, 59.389, -77.411, 67.099, 97.215, 16.558]
  MoveL 5292 to (232.37, 162.9, 78.65) mm, rotated rx 180 ry 0 rz 180 deg; joints [-66.048, 59.389, -77.411, 67.099, 97.215, 16.558]
  Call Extruder(269.35875)
  MoveL 5293 to (232.07, 163.03, 78.65) mm, rotated rx -180 ry 0 rz -180 deg; joints [-66.149, 59.389, -77.411, 67.197, 97.187, 16.571]
  MoveL 5294 to (232.07, 163.03, 78.65) mm, rotated rx -180 ry 0 rz -180 deg; joints [-66.149, 59.389, -77.411, 67.197, 97.187, 16.571]
  Call Extruder(269.54073)
  MoveL 5295 to (231.78, 163.15, 78.65) mm, rotated rx -180 ry 0 rz 180 deg; joints [-66.251, 59.388, -77.411, 67.295, 97.158, 16.584]
  MoveL 5296 to (231.78, 163.15, 78.65) mm, rotated rx -180 ry 0 rz 180 deg; joints [-66.251, 59.388, -77.411, 67.295, 97.158, 16.584]
  Call Extruder(269.68807)
  MoveL 5297 to (231.54, 163.24, 78.65) mm, rotated rx -180 ry 0 rz 180 deg; joints [-66.333, 59.387, -77.412, 67.375, 97.135, 16.596]
  MoveL 5298 to (231.54, 163.24, 78.65) mm, rotated rx -180 ry 0 rz 180 deg; joints [-66.333, 59.387, -77.412, 67.375, 97.135, 16.596]
  Call Extruder(269.80129)
  MoveL 5299 to (231.35, 163.3, 78.65) mm, rotated rx -180 ry 0 rz -180 deg; joints [-66.397, 59.386, -77.413, 67.437, 97.118, 16.605]
  MoveL 5300 to (231.35, 163.3, 78.65) mm, rotated rx -180 ry 0 rz -180 deg; joints [-66.397, 59.386, -77.413, 67.437, 97.118, 16.605]
  Call Extruder(269.91407)
  MoveL 5301 to (231.17, 163.36, 78.65) mm, rotated rx -180 ry 0 rz -180 deg; joints [-66.46, 59.384, -77.413, 67.498, 97.101, 16.615]
  MoveL 5302 to (231.17, 163.36, 78.65) mm, rotated rx -180 ry 0 rz -180 deg; joints [-66.46, 59.384, -77.413, 67.498, 97.101, 16.615]
  Call Extruder(270.02640)
  MoveL 5303 to (230.98, 163.42, 78.65) mm, rotated rx -180 ry 0 rz 180 deg; joints [-66.524, 59.382, -77.414, 67.56, 97.083, 16.625]
  MoveL 5304 to (230.98, 163.42, 78.65) mm, rotated rx -180 ry 0 rz 180 deg; joints [-66.524, 59.382, -77.414, 67.56, 97.083, 16.625]
  Call Extruder(270.13829)
  MoveL 5305 to (230.79, 163.48, 78.65) mm, rotated rx 180 ry 0 rz 180 deg; joints [-66.587, 59.381, -77.415, 67.621, 97.066, 16.635]
  MoveL 5306 to (230.79, 163.48, 78.65) mm, rotated rx 180 ry 0 rz 180 deg; joints [-66.587, 59.381, -77.415, 67.621, 97.066, 16.635]
  Call Extruder(270.25969)
  MoveL 5307 to (230.58, 163.55, 78.65) mm, rotated rx 180 ry 0 rz -180 deg; joints [-66.656, 59.379, -77.416, 67.688, 97.047, 16.645]
  MoveL 5308 to (230.58, 163.55, 78.65) mm, rotated rx 180 ry 0 rz -180 deg; joints [-66.656, 59.379, -77.416, 67.688, 97.047, 16.645]
  Call Extruder(270.39051)
  MoveL 5309 to (230.36, 163.62, 78.65) mm, rotated rx 180 ry 0 rz 180 deg; joints [-66.731, 59.377, -77.417, 67.761, 97.027, 16.657]
  MoveL 5310 to (230.36, 163.62, 78.65) mm, rotated rx 180 ry 0 rz 180 deg; joints [-66.731, 59.377, -77.417, 67.761, 97.027, 16.657]
  Call Extruder(270.52075)
  MoveL 5311 to (230.14, 163.68, 78.65) mm, rotated rx -180 ry 0 rz 180 deg; joints [-66.805, 59.375, -77.418, 67.833, 97.007, 16.669]
  MoveL 5312 to (230.14, 163.68, 78.65) mm, rotated rx -180 ry 0 rz 180 deg; joints [-66.805, 59.375, -77.418, 67.833, 97.007, 16.669]
  Call Extruder(270.65044)
  MoveL 5313 to (229.91, 163.75, 78.65) mm, rotated rx -180 ry 0 rz -180 deg; joints [-66.88, 59.373, -77.419, 67.906, 96.987, 16.68]
  MoveL 5314 to (229.91, 163.75, 78.65) mm, rotated rx -180 ry 0 rz -180 deg; joints [-66.88, 59.373, -77.419, 67.906, 96.987, 16.68]
  Call Extruder(270.77955)
  MoveL 5315 to (229.69, 163.82, 78.65) mm, rotated rx -180 ry 0 rz 180 deg; joints [-66.955, 59.371, -77.42, 67.978, 96.966, 16.692]
  MoveL 5316 to (229.69, 163.82, 78.65) mm, rotated rx -180 ry 0 rz 180 deg; joints [-66.955, 59.371, -77.42, 67.978, 96.966, 16.692]
  Call Extruder(270.89463)
  MoveL 5317 to (229.48, 163.86, 78.65) mm, rotated rx -180 ry 0 rz -180 deg; joints [-67.021, 59.368, -77.421, 68.043, 96.949, 16.704]
  MoveL 5318 to (229.48, 163.86, 78.65) mm, rotated rx -180 ry 0 rz -180 deg; joints [-67.021, 59.368, -77.421, 68.043, 96.949, 16.704]
  Call Extruder(271.00925)
  MoveL 5319 to (229.28, 163.91, 78.65) mm, rotated rx 180 ry 0 rz 180 deg; joints [-67.087, 59.365, -77.423, 68.107, 96.932, 16.716]
  MoveL 5320 to (229.28, 163.91, 78.65) mm, rotated rx 180 ry 0 rz 180 deg; joints [-67.087, 59.365, -77.423, 68.107, 96.932, 16.716]
  Call Extruder(271.12342)
  MoveL 5321 to (229.08, 163.95, 78.65) mm, rotated rx -180 ry 0 rz 180 deg; joints [-67.153, 59.362, -77.424, 68.171, 96.914, 16.728]
  MoveL 5322 to (229.08, 163.95, 78.65) mm, rotated rx -180 ry 0 rz 180 deg; joints [-67.153, 59.362, -77.424, 68.171, 96.914, 16.728]
  Call Extruder(271.23713)
  MoveL 5323 to (228.87, 164, 78.65) mm, rotated rx -180 ry 0 rz 180 deg; joints [-67.22, 59.359, -77.426, 68.236, 96.897, 16.74]
  MoveL 5324 to (228.87, 164, 78.65) mm, rotated rx -180 ry 0 rz 180 deg; joints [-67.22, 59.359, -77.426, 68.236, 96.897, 16.74]
  Call Extruder(271.36255)
  MoveL 5325 to (228.64, 164.04, 78.65) mm, rotated rx -180 ry 0 rz -180 deg; joints [-67.293, 59.355, -77.428, 68.307, 96.878, 16.753]
  MoveL 5326 to (228.64, 164.04, 78.65) mm, rotated rx -180 ry 0 rz -180 deg; joints [-67.293, 59.355, -77.428, 68.307, 96.878, 16.753]
  Call Extruder(271.49953)
  MoveL 5327 to (228.4, 164.09, 78.65) mm, rotated rx -180 ry 0 rz 180 deg; joints [-67.373, 59.351, -77.429, 68.385, 96.857, 16.768]
  MoveL 5328 to (228.4, 164.09, 78.65) mm, rotated rx -180 ry 0 rz 180 deg; joints [-67.373, 59.351, -77.429, 68.385, 96.857, 16.768]
  Call Extruder(271.63590)
  MoveL 5329 to (228.15, 164.14, 78.65) mm, rotated rx -180 ry 0 rz 180 deg; joints [-67.453, 59.347, -77.431, 68.463, 96.836, 16.783]
  MoveL 5330 to (228.15, 164.14, 78.65) mm, rotated rx -180 ry 0 rz 180 deg; joints [-67.453, 59.347, -77.431, 68.463, 96.836, 16.783]
  Call Extruder(271.77166)
  MoveL 5331 to (227.9, 164.19, 78.65) mm, rotated rx -180 ry 0 rz -180 deg; joints [-67.534, 59.343, -77.433, 68.541, 96.815, 16.797]
  MoveL 5332 to (227.9, 164.19, 78.65) mm, rotated rx -180 ry 0 rz -180 deg; joints [-67.534, 59.343, -77.433, 68.541, 96.815, 16.797]
  Call Extruder(271.90680)
  MoveL 5333 to (227.65, 164.24, 78.65) mm, rotated rx 180 ry 0 rz -180 deg; joints [-67.614, 59.339, -77.435, 68.619, 96.794, 16.812]
  MoveL 5334 to (227.65, 164.24, 78.65) mm, rotated rx 180 ry 0 rz -180 deg; joints [-67.614, 59.339, -77.435, 68.619, 96.794, 16.812]
  Call Extruder(272.04134)
  MoveL 5335 to (227.4, 164.29, 78.65) mm, rotated rx -180 ry 0 rz 180 deg; joints [-67.695, 59.335, -77.437, 68.697, 96.773, 16.827]
  MoveL 5336 to (227.4, 164.29, 78.65) mm, rotated rx -180 ry 0 rz 180 deg; joints [-67.695, 59.335, -77.437, 68.697, 96.773, 16.827]
  Call Extruder(272.17527)
  MoveL 5337 to (227.15, 164.34, 78.65) mm, rotated rx -180 ry 0 rz -180 deg; joints [-67.775, 59.331, -77.439, 68.775, 96.751, 16.841]
  MoveL 5338 to (227.15, 164.34, 78.65) mm, rotated rx -180 ry 0 rz -180 deg; joints [-67.775, 59.331, -77.439, 68.775, 96.751, 16.841]
  Call Extruder(272.32313)
  MoveL 5339 to (226.87, 164.39, 78.65) mm, rotated rx -180 ry 0 rz 180 deg; joints [-67.864, 59.327, -77.441, 68.862, 96.728, 16.858]
  MoveL 5340 to (226.87, 164.39, 78.65) mm, rotated rx -180 ry 0 rz 180 deg; joints [-67.864, 59.327, -77.441, 68.862, 96.728, 16.858]
  Call Extruder(272.48487)
  MoveL 5341 to (226.57, 164.44, 78.65) mm, rotated rx 180 ry 0 rz -180 deg; joints [-67.961, 59.321, -77.444, 68.957, 96.703, 16.877]
  MoveL 5342 to (226.57, 164.44, 78.65) mm, rotated rx 180 ry 0 rz -180 deg; joints [-67.961, 59.321, -77.444, 68.957, 96.703, 16.877]
  Call Extruder(272.64589)
  MoveL 5343 to (226.26, 164.49, 78.65) mm, rotated rx 180 ry 0 rz 180 deg; joints [-68.059, 59.315, -77.447, 69.051, 96.678, 16.895]
  MoveL 5344 to (226.26, 164.49, 78.65) mm, rotated rx 180 ry 0 rz 180 deg; joints [-68.059, 59.315, -77.447, 69.051, 96.678, 16.895]
  Call Extruder(272.80617)
  MoveL 5345 to (225.96, 164.53, 78.65) mm, rotated rx 180 ry 0 rz 180 deg; joints [-68.156, 59.31, -77.449, 69.146, 96.652, 16.914]
  MoveL 5346 to (225.96, 164.53, 78.65) mm, rotated rx 180 ry 0 rz 180 deg; joints [-68.156, 59.31, -77.449, 69.146, 96.652, 16.914]
  Call Extruder(272.96573)
  MoveL 5347 to (225.65, 164.58, 78.65) mm, rotated rx 180 ry 0 rz 180 deg; joints [-68.254, 59.304, -77.452, 69.241, 96.627, 16.933]
  MoveL 5348 to (225.65, 164.58, 78.65) mm, rotated rx 180 ry 0 rz 180 deg; joints [-68.254, 59.304, -77.452, 69.241, 96.627, 16.933]
  Call Extruder(273.12456)
  MoveL 5349 to (225.34, 164.63, 78.65) mm, rotated rx -180 ry 0 rz 180 deg; joints [-68.351, 59.299, -77.455, 69.336, 96.601, 16.951]
  MoveL 5350 to (225.34, 164.63, 78.65) mm, rotated rx -180 ry 0 rz 180 deg; joints [-68.351, 59.299, -77.455, 69.336, 96.601, 16.951]
  Call Extruder(273.30323)
  MoveL 5351 to (225, 164.68, 78.65) mm, rotated rx 180 ry 0 rz -180 deg; joints [-68.461, 59.292, -77.458, 69.443, 96.572, 16.973]
  MoveL 5352 to (225, 164.68, 78.65) mm, rotated rx 180 ry 0 rz -180 deg; joints [-68.461, 59.292, -77.458, 69.443, 96.572, 16.973]
  Call Extruder(273.50167)
  MoveL 5353 to (224.61, 164.73, 78.65) mm, rotated rx -180 ry 0 rz 180 deg; joints [-68.583, 59.284, -77.462, 69.562, 96.541, 16.997]
  MoveL 5354 to (224.61, 164.73, 78.65) mm, rotated rx -180 ry 0 rz 180 deg; joints [-68.583, 59.284, -77.462, 69.562, 96.541, 16.997]
  Call Extruder(273.69925)
  MoveL 5355 to (224.22, 164.77, 78.65) mm, rotated rx 180 ry 0 rz 180 deg; joints [-68.706, 59.276, -77.466, 69.681, 96.509, 17.021]
  MoveL 5356 to (224.22, 164.77, 78.65) mm, rotated rx 180 ry 0 rz 180 deg; joints [-68.706, 59.276, -77.466, 69.681, 96.509, 17.021]
  Call Extruder(273.89595)
  MoveL 5357 to (223.84, 164.82, 78.65) mm, rotated rx 180 ry 0 rz -180 deg; joints [-68.828, 59.269, -77.469, 69.8, 96.477, 17.046]
  MoveL 5358 to (223.84, 164.82, 78.65) mm, rotated rx 180 ry 0 rz -180 deg; joints [-68.828, 59.269, -77.469, 69.8, 96.477, 17.046]
  Call Extruder(274.09179)
  MoveL 5359 to (223.45, 164.86, 78.65) mm, rotated rx -180 ry 0 rz 180 deg; joints [-68.951, 59.261, -77.473, 69.919, 96.445, 17.07]
  MoveL 5360 to (223.45, 164.86, 78.65) mm, rotated rx -180 ry 0 rz 180 deg; joints [-68.951, 59.261, -77.473, 69.919, 96.445, 17.07]
  Call Extruder(274.38715)
  MoveL 5361 to (222.86, 164.91, 78.65) mm, rotated rx -180 ry 0 rz 180 deg; joints [-69.135, 59.247, -77.479, 70.098, 96.398, 17.108]
  MoveL 5362 to (222.86, 164.91, 78.65) mm, rotated rx -180 ry 0 rz 180 deg; joints [-69.135, 59.247, -77.479, 70.098, 96.398, 17.108]
  Call Extruder(274.68118)
  MoveL 5363 to (222.27, 164.95, 78.65) mm, rotated rx -180 ry 0 rz 180 deg; joints [-69.319, 59.234, -77.486, 70.277, 96.35, 17.147]
  MoveL 5364 to (222.27, 164.95, 78.65) mm, rotated rx -180 ry 0 rz 180 deg; joints [-69.319, 59.234, -77.486, 70.277, 96.35, 17.147]
  Call Extruder(274.97387)
  MoveL 5365 to (221.68, 165, 78.65) mm, rotated rx -180 ry 0 rz 180 deg; joints [-69.504, 59.221, -77.492, 70.457, 96.302, 17.185]
  MoveL 5366 to (221.68, 165, 78.65) mm, rotated rx -180 ry 0 rz 180 deg; joints [-69.504, 59.221, -77.492, 70.457, 96.302, 17.185]
  Call Extruder(275.54732)
  MoveL 5367 to (220.52, 165.05, 78.65) mm, rotated rx -180 ry 0 rz 180 deg; joints [-69.864, 59.192, -77.506, 70.807, 96.21, 17.263]
  MoveL 5368 to (220.52, 165.05, 78.65) mm, rotated rx -180 ry 0 rz 180 deg; joints [-69.864, 59.192, -77.506, 70.807, 96.21, 17.263]
  Call Extruder(276.26133)
  MoveL 5369 to (219.06, 165.09, 78.65) mm, rotated rx -180 ry 0 rz 180 deg; joints [-70.315, 59.155, -77.523, 71.246, 96.093, 17.361]
  Call Extruder(393.10807)
  MoveL 5370 to (-19.06, 165.09, 78.65) mm, rotated rx 180 ry 0 rz 180 deg; joints [-137.325, 63.978, -74.051, 136.881, 82.612, 6.866]
  Call Extruder(393.53667)
  MoveL 5371 to (-19.94, 165.07, 78.65) mm, rotated rx 180 ry 0 rz 180 deg; joints [-137.467, 64.016, -74.011, 137.031, 82.652, 6.794]
  MoveL 5372 to (-19.94, 165.07, 78.65) mm, rotated rx 180 ry 0 rz 180 deg; joints [-137.467, 64.016, -74.011, 137.031, 82.652, 6.794]
  Call Extruder(394.11012)
  MoveL 5373 to (-21.1, 165.02, 78.65) mm, rotated rx -180 ry 0 rz 180 deg; joints [-137.659, 64.066, -73.958, 137.231, 82.705, 6.699]
  MoveL 5374 to (-21.1, 165.02, 78.65) mm, rotated rx -180 ry 0 rz 180 deg; joints [-137.659, 64.066, -73.958, 137.231, 82.705, 6.699]
  Call Extruder(394.54442)
  MoveL 5375 to (-21.97, 164.98, 78.65) mm, rotated rx 180 ry 0 rz 180 deg; joints [-137.804, 64.103, -73.918, 137.384, 82.745, 6.628]
